		IF uiCommandDoneNum = stAdvHomePara_Set.uiCommandNum THEN//All commands are done
			
			iStep_Homing:=10000;//Done Step
		ELSE
			
			IF uiCommandDoneNum > 0 THEN
				uiCurrentCmdNo:=uiCurrentCmdNo+1;
			END_IF
			
			iStep_Homing:=300;
		END_IF

	300://Decide Step Function and Set Parameter
	
		//Get Homing Para From [SET]
		stAdvHomePara_Local:=stAdvHomePara_Set;
		
		//Set Speed According to Command List content
		IF stAdvHomePara_Local.stHomingCommand[uiCurrentCmdNo].bSlowVelo THEN
			stAdvHomePara_Local.stHomingCommand[uiCurrentCmdNo].stStepFuncParameter.MovePara			:=MovePara_Slow;
			stAdvHomePara_Local.stHomingCommand[uiCurrentCmdNo].stStepFuncParameter.stHomingLimitation	:=MoveLimitation_Slow;
		ELSE
			stAdvHomePara_Local.stHomingCommand[uiCurrentCmdNo].stStepFuncParameter.MovePara			:=MovePara_Fast;
			stAdvHomePara_Local.stHomingCommand[uiCurrentCmdNo].stStepFuncParameter.stHomingLimitation	:=MoveLimitation_Fast;
		END_IF
		
		//Get Homing Function Action Type
		eHome_ActionType:=stAdvHomePara_Local.stHomingCommand[uiCurrentCmdNo].eHome_ActionType;
		
		//Flag On
		IF eHome_ActionType = E_HomingActionType.FinishHoming
		OR eHome_ActionType = E_HomingActionType.HomeDirect 
		THEN
			iStep_FinalizingFunc:=1;
		ELSIF eHome_ActionType = E_HomingActionType.ParameterSetting THEN
			iStep_ParaSetting:=1;
		ELSE
			iStep_StepFunc:=1;
		END_IF
		
		iStep_Homing:=400;
		
	400://Step/Finalizing/Parameter Function
		CASE eHome_ActionType OF
			(* ---------- Step Function ----------*)
			E_HomingActionType.Dog_Abs:
				IF M_DogAbs(stAdvHomePara_Local.stHomingCommand[uiCurrentCmdNo].stStepFuncParameter,lrSetPosition,ErrorId=>uiStepFuncErrorId) THEN
					IF uiStepFuncErrorId = 0 THEN
						uiCommandDoneNum:=uiCommandDoneNum+1;
						iStep_Homing:=200;
					ELSE
						iStep_Homing:=9001;
					END_IF
				END_IF
			E_HomingActionType.Dog_Detection:
				IF M_DogDetection(stAdvHomePara_Local.stHomingCommand[uiCurrentCmdNo].stStepFuncParameter,ErrorId=>uiStepFuncErrorId) THEN
					IF uiStepFuncErrorId = 0 THEN
						uiCommandDoneNum:=uiCommandDoneNum+1;
						iStep_Homing:=200;
					ELSE
						iStep_Homing:=9002;
					END_IF
				END_IF
			E_HomingActionType.Index_Abs:
				IF M_PulseFind(stAdvHomePara_Local.stHomingCommand[uiCurrentCmdNo].stStepFuncParameter,lrSetPosition,ErrorId=>uiStepFuncErrorId) THEN
					IF uiStepFuncErrorId = 0 THEN
						uiCommandDoneNum:=uiCommandDoneNum+1;
						iStep_Homing:=200;
					ELSE
						iStep_Homing:=9003;
					END_IF
				END_IF
			E_HomingActionType.Index_Detection:
				IF M_PulseDetection(stAdvHomePara_Local.stHomingCommand[uiCurrentCmdNo].stStepFuncParameter,ErrorId=>uiStepFuncErrorId) THEN
					IF uiStepFuncErrorId = 0 THEN
						uiCommandDoneNum:=uiCommandDoneNum+1;
						iStep_Homing:=200;
					ELSE
						iStep_Homing:=9004;
					END_IF
				END_IF
			E_HomingActionType.Limit_Abs:
				//Set Ref Switch Signal
				IF stAdvHomePara_Local.bRefNegLimitSignal THEN
					fbStepLimitSwitch.LimitSwitchSignal:=NegLimitSwitchSignal;
				ELSE
					fbStepLimitSwitch.LimitSwitchSignal:=PosLimitSwitchSignal;
				END_IF
				
				IF M_LimitFind(stAdvHomePara_Local.stHomingCommand[uiCurrentCmdNo].stStepFuncParameter,lrSetPosition,ErrorId=>uiStepFuncErrorId) THEN
					IF uiStepFuncErrorId = 0 THEN
						uiCommandDoneNum:=uiCommandDoneNum+1;
						iStep_Homing:=200;
					ELSE
						iStep_Homing:=9005;
					END_IF
				END_IF
			E_HomingActionType.Limit_Detection:
				//Set Ref Switch Signal
				IF stAdvHomePara_Local.bRefNegLimitSignal THEN
					fbStepLimitSwitchDetection.LimitSwitchSignal:=NegLimitSwitchSignal;
				ELSE
					fbStepLimitSwitchDetection.LimitSwitchSignal:=PosLimitSwitchSignal;
				END_IF
				
				IF M_LimitDetection(stAdvHomePara_Local.stHomingCommand[uiCurrentCmdNo].stStepFuncParameter,ErrorId=>uiStepFuncErrorId) THEN
					IF uiStepFuncErrorId = 0 THEN
						uiCommandDoneNum:=uiCommandDoneNum+1;
						iStep_Homing:=200;
					ELSE
						iStep_Homing:=9006;
					END_IF
				END_IF
			(* ---------- Finish Function ----------*)
			E_HomingActionType.FinishHoming:
				IF M_FinishHoming(stAdvHomePara_Local.stHomingCommand[uiCurrentCmdNo].stStepFuncParameter,lrOffset) THEN
					uiCommandDoneNum:=uiCommandDoneNum+1;
					iStep_Homing:=200;
				END_IF
			E_HomingActionType.HomeDirect:
				IF M_HomeDirect(stAdvHomePara_Local.stHomingCommand[uiCurrentCmdNo].stStepFuncParameter,lrSetPosition) THEN
					uiCommandDoneNum:=uiCommandDoneNum+1;
					iStep_Homing:=200;
				END_IF
			(* ---------- Parameter Function ----------*)	
			E_HomingActionType.ParameterSetting:
				IF M_KeepPosBias(stPosBiasPara.bModuloMode,lrSetPosition) THEN
					uiCommandDoneNum:=uiCommandDoneNum+1;
					iStep_Homing:=200;
				END_IF
			E_HomingActionType.MoveAbs:
				IF M_MoveAbs(stAdvHomePara_Local.stHomingCommand[uiCurrentCmdNo].stStepFuncParameter,lrSetPosition) THEN
					IF uiStepFuncErrorId = 0 THEN
						uiCommandDoneNum:=uiCommandDoneNum+1;
						iStep_Homing:=200;
					ELSE
						iStep_Homing:=9007;
					END_IF
				END_IF
			ELSE//Not Defined Action Type
				ErrorId:=400;
				iStep_Homing:=9000;//Error Step
		END_CASE
	
	(*-----Aborting-----*)
	8000://Abort
	
		iStep_FinalizingFunc:=1;
		
		iStep_Homing:=8100;
	8100:
		IF M_AbortHoming() THEN
			iStep_Homing:=10000;
		END_IF
	9000:
		M_SetError(ErrorId);
	(*-----Step Func Error-----*)
	9001..9099:(* Abort *)
		iStep_FinalizingFunc:=1;
		iStep_Homing:=iStep_Homing+100;
	9101..9199:
		IF M_AbortHoming() THEN
			M_SetError(uiStepFuncErrorId);
			iStep_Homing:=iStep_Homing+100;
		END_IF
	(*-----Done-----*)
	10000://Done
		M_SetDone();
		iStep_Homing:=10100;
END_CASE

METHOD PRIVATE M_ClearAllState : BOOL
VAR_INPUT
END_VAR
fbStepAbsoluteSwitchDetection.Execute 	:= FALSE;
fbStepAbsoluteSwitch.Execute 			:= FALSE;				
fbStepLimitSwitchDetection.Execute 		:= FALSE;			
fbStepLimitSwitch.Execute 				:= FALSE;					
fbStepReferencePulse.Execute 			:= FALSE;
fbStepReferencePulseDetection.Execute 	:= FALSE;
fbFinishHoming.Execute					:= FALSE;
fbHomeDirect.Execute					:= FALSE;
fbAbortHoming.Execute 					:= FALSE;

uiCurrentCmdNo:=0;
uiCommandDoneNum:=0;
	
iStep_FinalizingFunc:=0;
iStep_StepFunc:=0;

iStep_Homing:=0;
END_METHOD

METHOD PRIVATE M_ClearSignal : BOOL
VAR_INPUT
END_VAR
Done			:=FALSE;
Busy 			:=FALSE;
Active   		:=FALSE;
CommandAborted	:=FALSE;
Error			:=FALSE;
ErrorId 		:=0;
END_METHOD

METHOD private M_SetBusy : BOOL
VAR_INPUT
END_VAR
M_ClearSignal();

Busy:=TRUE;
END_METHOD

METHOD private M_SetDone : BOOL
VAR_INPUT
END_VAR
M_ClearSignal();

Done:=TRUE;
END_METHOD

METHOD PRIVATE M_SetError : BOOL
VAR_INPUT
	setErrorId:UDINT;
END_VAR
M_ClearSignal();

Error := TRUE;
ErrorId := setErrorId;
END_METHOD

METHOD PRIVATE M_DogAbs : BOOL
VAR_INPUT
	stStepFuncParameter		:ST_StepFuncParameter;
	SetPosition				:LREAL;
END_VAR
VAR_OUTPUT
	ErrorId		:UDINT:=0;
END_VAR
CASE iStep_StepFunc	OF
	1:
		fbStepAbsoluteSwitch.Direction			:= stStepFuncParameter.eHome_Direction;
		fbStepAbsoluteSwitch.SwitchMode		    := stStepFuncParameter.eSwitch_Mode;
		
		fbStepAbsoluteSwitch.Velocity			:= stStepFuncParameter.MovePara.Velocity;
		fbStepAbsoluteSwitch.Acceleration		:= stStepFuncParameter.MovePara.Acc;
		fbStepAbsoluteSwitch.Deceleration		:= stStepFuncParameter.MovePara.Dec;
		fbStepAbsoluteSwitch.Jerk				:= stStepFuncParameter.MovePara.Jerk;
		
		fbStepAbsoluteSwitch.TimeLimit			:= stStepFuncParameter.stHomingLimitation.TimeLimit;
		fbStepAbsoluteSwitch.DistanceLimit		:= stStepFuncParameter.stHomingLimitation.DistanceLimit;
		fbStepAbsoluteSwitch.TorqueLimit		:= stStepFuncParameter.stHomingLimitation.TorqueLimit;
		
		fbStepAbsoluteSwitch.SetPosition		:= SetPosition;
		
		fbStepAbsoluteSwitch.Execute 			:= TRUE;
		
		IF	fbStepAbsoluteSwitch.Busy	THEN
			iStep_StepFunc:= 2;
		END_IF
	
	2:
		IF	fbStepAbsoluteSwitch.Done	THEN
			fbStepAbsoluteSwitch.Execute 		:= FALSE;
			iStep_StepFunc:= 3;	
		ELSIF fbStepAbsoluteSwitch.Error	THEN
			iStep_StepFunc:= 90;
		END_IF
	3:
		iStep_StepFunc:=0;
		M_DogAbs:=TRUE;
	(* Error *)
	90:
		ErrorId:=fbStepAbsoluteSwitch.ErrorID;
		
		fbStepAbsoluteSwitch.Execute:=FALSE;
		M_DogAbs:=TRUE;
END_CASE
END_METHOD

METHOD PRIVATE M_DogDetection : BOOL
VAR_INPUT
	stStepFuncParameter		:ST_StepFuncParameter;
END_VAR
VAR_OUTPUT
	ErrorId		:UDINT:=0;
END_VAR
CASE iStep_StepFunc	OF
	1:
		fbStepAbsoluteSwitchDetection.Direction			:= stStepFuncParameter.eHome_Direction;
		fbStepAbsoluteSwitchDetection.SwitchMode		:= stStepFuncParameter.eSwitch_Mode;
		
		fbStepAbsoluteSwitchDetection.Velocity			:= stStepFuncParameter.MovePara.Velocity;
		fbStepAbsoluteSwitchDetection.Acceleration		:= stStepFuncParameter.MovePara.Acc;
		fbStepAbsoluteSwitchDetection.Deceleration		:= stStepFuncParameter.MovePara.Dec;
		fbStepAbsoluteSwitchDetection.Jerk				:= stStepFuncParameter.MovePara.Jerk;
		
		fbStepAbsoluteSwitchDetection.TimeLimit			:= stStepFuncParameter.stHomingLimitation.TimeLimit;
		fbStepAbsoluteSwitchDetection.DistanceLimit		:= stStepFuncParameter.stHomingLimitation.DistanceLimit;
		fbStepAbsoluteSwitchDetection.TorqueLimit		:= stStepFuncParameter.stHomingLimitation.TorqueLimit;
		
		fbStepAbsoluteSwitchDetection.Execute 			:= TRUE;
		
		IF	fbStepAbsoluteSwitchDetection.Busy	THEN
			iStep_StepFunc:= 2;
		END_IF
	
	2:
		IF	fbStepAbsoluteSwitchDetection.Done	THEN
			fbStepAbsoluteSwitchDetection.Execute 		:= FALSE;
			iStep_StepFunc:= 3;	
		ELSIF fbStepAbsoluteSwitchDetection.Error THEN
			iStep_StepFunc:= 90;
		END_IF
	3:
		iStep_StepFunc:=0;
		M_DogDetection:=TRUE;
	(* Error *)
	90:
		ErrorId:=fbStepAbsoluteSwitchDetection.ErrorID;
		
		fbStepAbsoluteSwitchDetection.Execute:=FALSE;
		M_DogDetection:=TRUE;
END_CASE
END_METHOD

METHOD PRIVATE M_LimitDetection : BOOL
VAR_INPUT
	stStepFuncParameter		:ST_StepFuncParameter;
END_VAR
VAR_OUTPUT
	ErrorId		:UDINT:=0;
END_VAR
CASE iStep_StepFunc	OF
	1:
		fbStepLimitSwitchDetection.Direction			:= stStepFuncParameter.eHome_Direction;
		fbStepLimitSwitchDetection.LimitSwitchMode		:= stStepFuncParameter.eSwitch_Mode;
		
		fbStepLimitSwitchDetection.Velocity			:= stStepFuncParameter.MovePara.Velocity;
		fbStepLimitSwitchDetection.Acceleration		:= stStepFuncParameter.MovePara.Acc;
		fbStepLimitSwitchDetection.Deceleration		:= stStepFuncParameter.MovePara.Dec;
		fbStepLimitSwitchDetection.Jerk				:= stStepFuncParameter.MovePara.Jerk;
		
		fbStepLimitSwitchDetection.TimeLimit		:= stStepFuncParameter.stHomingLimitation.TimeLimit;
		fbStepLimitSwitchDetection.DistanceLimit	:= stStepFuncParameter.stHomingLimitation.DistanceLimit;
		fbStepLimitSwitchDetection.TorqueLimit		:= stStepFuncParameter.stHomingLimitation.TorqueLimit;
		
		fbStepLimitSwitchDetection.Execute := TRUE;
		
		IF	fbStepLimitSwitchDetection.Busy	THEN
			iStep_StepFunc:= 2;
		END_IF
	
	2:
		IF	fbStepLimitSwitchDetection.Done	THEN
			fbStepLimitSwitchDetection.Execute := FALSE;
			iStep_StepFunc:= 3;	
		ELSIF fbStepLimitSwitchDetection.Error THEN
			iStep_StepFunc:= 90;	
		END_IF
	3:
		iStep_StepFunc:=0;
		M_LimitDetection:=TRUE;
	(* Error *)
	90:
		ErrorId:=fbStepLimitSwitchDetection.ErrorID;
		
		fbStepLimitSwitchDetection.Execute:=FALSE;
		M_LimitDetection:=TRUE;
END_CASE
END_METHOD

METHOD PRIVATE M_LimitFind : BOOL
VAR_INPUT
	stStepFuncParameter		:ST_StepFuncParameter;
	SetPosition				:LREAL;
END_VAR
VAR_OUTPUT
	ErrorId		:UDINT:=0;
END_VAR
CASE iStep_StepFunc	OF
	1://拉起找極限
		fbStepLimitSwitch.Direction			:= stStepFuncParameter.eHome_Direction;
		fbStepLimitSwitch.LimitSwitchMode		:= stStepFuncParameter.eSwitch_Mode;
		
		fbStepLimitSwitch.Velocity			:= stStepFuncParameter.MovePara.Velocity;
		fbStepLimitSwitch.Acceleration		:= stStepFuncParameter.MovePara.Acc;
		fbStepLimitSwitch.Deceleration		:= stStepFuncParameter.MovePara.Dec;
		fbStepLimitSwitch.Jerk				:= stStepFuncParameter.MovePara.Jerk;
		
		fbStepLimitSwitch.TimeLimit			:= stStepFuncParameter.stHomingLimitation.TimeLimit;
		fbStepLimitSwitch.DistanceLimit		:= stStepFuncParameter.stHomingLimitation.DistanceLimit;
		fbStepLimitSwitch.TorqueLimit		:= stStepFuncParameter.stHomingLimitation.TorqueLimit;
		
		fbStepLimitSwitch.SetPosition		:= SetPosition;
		
		fbStepLimitSwitch.Execute := TRUE;
		
		IF	fbStepLimitSwitch.Busy	THEN
			iStep_StepFunc:= 2;
		END_IF
	
	2://等待完成
		IF	fbStepLimitSwitch.Done	THEN
			fbStepLimitSwitch.Execute:= FALSE;
			iStep_StepFunc:= 3;	
		ELSIF fbStepLimitSwitch.Error THEN
			iStep_StepFunc:= 90;	
		END_IF
	3://完成處理
		iStep_StepFunc:=0;
		M_LimitFind:=TRUE;
	(* Error *)
	90:
		ErrorId:=fbStepLimitSwitch.ErrorID;
		
		fbStepLimitSwitch.Execute:=FALSE;
		M_LimitFind:=TRUE;
END_CASE
END_METHOD

METHOD M_MoveAbs : BOOL
VAR_INPUT
	stStepFuncParameter		:ST_StepFuncParameter;
	SetPosition				:LREAL;
END_VAR
VAR_OUTPUT
	ErrorId		:UDINT:=0;
END_VAR
CASE iStep_StepFunc OF
    1:
        fbMoveAbs.Acceleration := stStepFuncParameter.MovePara.Acc;
        fbMoveAbs.Deceleration := stStepFuncParameter.MovePara.Dec;
        fbMoveAbs.Jerk := stStepFuncParameter.MovePara.Jerk;
        fbMoveAbs.Velocity := stStepFuncParameter.MovePara.Velocity;
        fbMoveAbs.Position := SetPosition;
		fbMoveAbs.Execute := TRUE;
        IF fbMoveAbs.Busy THEN
            iStep_StepFunc := 2;
        END_IF

    2:
        IF fbMoveAbs.Done THEN
            fbMoveAbs.Execute := FALSE;
            iStep_StepFunc := 3;
        ELSIF fbMoveAbs.Error THEN
            iStep_StepFunc := 90;
        END_IF
    3:
        iStep_StepFunc := 0;
        M_MoveAbs := TRUE;
        (* Error *)
        ErrorId := fbMoveAbs.ErrorID;

        fbMoveAbs.Execute := FALSE;
        M_MoveAbs := TRUE;

END_CASE
END_METHOD

METHOD PRIVATE M_PulseDetection : BOOL
VAR_INPUT
	stStepFuncParameter		:ST_StepFuncParameter;
END_VAR
VAR_OUTPUT
	ErrorId		:UDINT:=0;
END_VAR
CASE iStep_StepFunc	OF
	1:
		fbStepReferencePulseDetection.Direction			:= stStepFuncParameter.eHome_Direction;
		
		fbStepReferencePulseDetection.Velocity			:= stStepFuncParameter.MovePara.Velocity;
		fbStepReferencePulseDetection.Acceleration		:= stStepFuncParameter.MovePara.Acc;
		fbStepReferencePulseDetection.Deceleration		:= stStepFuncParameter.MovePara.Dec;
		fbStepReferencePulseDetection.Jerk				:= stStepFuncParameter.MovePara.Jerk;
		
		fbStepReferencePulseDetection.TimeLimit			:= stStepFuncParameter.stHomingLimitation.TimeLimit;
		fbStepReferencePulseDetection.DistanceLimit		:= stStepFuncParameter.stHomingLimitation.DistanceLimit;
		fbStepReferencePulseDetection.TorqueLimit		:= stStepFuncParameter.stHomingLimitation.TorqueLimit;
		
		fbStepReferencePulseDetection.Execute 			:= TRUE;
		
		IF	fbStepReferencePulseDetection.Busy	THEN
			iStep_StepFunc:= 2;
		END_IF
	
	2:
		IF	fbStepReferencePulseDetection.Done	THEN
			fbStepReferencePulseDetection.Execute 		:= FALSE;
			iStep_StepFunc:= 3;	
		ELSIF fbStepReferencePulseDetection.Error THEN
			iStep_StepFunc:= 90;	
		END_IF
	3:
		iStep_StepFunc:=0;
		M_PulseDetection:=TRUE;
	(* Error *)
	90:
		ErrorId:=fbStepReferencePulseDetection.ErrorID;
		
		fbStepReferencePulseDetection.Execute:=FALSE;
		M_PulseDetection:=TRUE;
END_CASE
END_METHOD

METHOD PRIVATE M_PulseFind : BOOL
VAR_INPUT
	stStepFuncParameter		:ST_StepFuncParameter;
	SetPosition				:LREAL;
END_VAR
VAR_OUTPUT
	ErrorId		:UDINT:=0;
END_VAR
CASE iStep_StepFunc OF 
	1://拉起找Zero Pulse
	
		fbStepReferencePulse.Direction			:= stStepFuncParameter.eHome_Direction;
		
		fbStepReferencePulse.Velocity			:= stStepFuncParameter.MovePara.Velocity;
		fbStepReferencePulse.Acceleration		:= stStepFuncParameter.MovePara.Acc;
		fbStepReferencePulse.Deceleration		:= stStepFuncParameter.MovePara.Dec;
		fbStepReferencePulse.Jerk				:= stStepFuncParameter.MovePara.Jerk;
		
		fbStepReferencePulse.TimeLimit			:= stStepFuncParameter.stHomingLimitation.TimeLimit;
		fbStepReferencePulse.DistanceLimit		:= stStepFuncParameter.stHomingLimitation.DistanceLimit;
		fbStepReferencePulse.TorqueLimit		:= stStepFuncParameter.stHomingLimitation.TorqueLimit;
		
		fbStepReferencePulse.SetPosition		:= SetPosition;
		
		fbStepReferencePulse.Execute 			:= TRUE;
		
		IF	fbStepReferencePulse.Busy THEN
			iStep_StepFunc:= 2;
		END_IF
	
	2:
		IF	fbStepReferencePulse.Done	THEN
			fbStepReferencePulse.Execute:= FALSE;
			iStep_StepFunc:= 3;
		ELSIF fbStepReferencePulse.Error THEN
			iStep_StepFunc:= 90;
		END_IF
	3:
		iStep_StepFunc:=0;
		M_PulseFind:=TRUE;
	(* Error *)
	90:
		ErrorId:=fbStepReferencePulse.ErrorID;
		
		fbStepReferencePulse.Execute:=FALSE;
		M_PulseFind:=TRUE;
END_CASE
END_METHOD

METHOD PRIVATE M_AbortHoming : BOOL
VAR_INPUT
END_VAR
CASE iStep_FinalizingFunc OF
	1:
		fbAbortHoming.Execute 					:= TRUE;
		
		IF	fbAbortHoming.Busy	THEN
			iStep_FinalizingFunc:= 2;
		END_IF
	2:
		IF	fbAbortHoming.Done	THEN
			fbAbortHoming.Execute 		:= FALSE;
			iStep_FinalizingFunc:= 3;	
		END_IF
	3:
		iStep_FinalizingFunc:=0;
		M_AbortHoming:=TRUE;
END_CASE
END_METHOD

METHOD PRIVATE M_FinishHoming : BOOL
VAR_INPUT
	stStepFuncParameter		:ST_StepFuncParameter;
	Distance				:LREAL;
END_VAR
CASE iStep_FinalizingFunc OF
	1:
		fbFinishHoming.Velocity			:= stStepFuncParameter.MovePara.Velocity;
		fbFinishHoming.Acceleration		:= stStepFuncParameter.MovePara.Acc;
		fbFinishHoming.Deceleration		:= stStepFuncParameter.MovePara.Dec;
		fbFinishHoming.Jerk				:= stStepFuncParameter.MovePara.Jerk;
		
		fbFinishHoming.Distance			:=Distance;
		
		fbFinishHoming.Execute 			:= TRUE;
		
		IF	fbFinishHoming.Busy	THEN
			iStep_FinalizingFunc:= 2;
		END_IF
	2:
		IF	fbFinishHoming.Done	THEN
			fbFinishHoming.Execute 		:= FALSE;
			iStep_FinalizingFunc:= 3;	
		END_IF
	3:
		iStep_FinalizingFunc:=0;
		M_FinishHoming:=TRUE;
END_CASE
END_METHOD

METHOD PRIVATE M_HomeDirect : BOOL
VAR_INPUT
	stStepFuncParameter		:ST_StepFuncParameter;
	SetPosition				:LREAL;
END_VAR
CASE iStep_FinalizingFunc OF
	1:
		fbHomeDirect.SetPosition:=SetPosition;
		
		fbHomeDirect.Execute:=TRUE;
		
		IF	fbHomeDirect.Busy	THEN
			iStep_FinalizingFunc:= 2;
		END_IF
	2:
		IF	fbHomeDirect.Done	THEN
			fbHomeDirect.Execute 		:= FALSE;
			iStep_FinalizingFunc:= 3;	
		END_IF
	3:
		iStep_FinalizingFunc:=0;
		M_HomeDirect:=TRUE;
END_CASE
END_METHOD

METHOD M_KeepPosBias : BOOL
VAR_INPUT
	bModuloMode		:BOOL:=FALSE;//True=Modulo Bias
	SetPosition		:LREAL;
END_VAR
VAR
	lrNcCurrentBias	:LREAL;
	lrNcCurrentPos	:LREAL;
	lrNcTargetPos	:LREAL;
	lrNcTargetBias	:LREAL;
	lrNcOriginPos	:LREAL;
END_VAR
CASE iStep_ParaSetting OF
	1://Read Current Bias Value
	
		fbReadParameter.Enable				:= TRUE;
		fbReadParameter.ReadMode			:= E_ReadMode.READMODE_ONCE;
		fbReadParameter.ParameterNumber		:= MC_AxisParameter.AxisEncoderOffset;//Position Bias
		
		IF fbReadParameter.Valid THEN
			fbReadParameter.Enable:=FALSE;
			iStep_ParaSetting:= 2;
		ELSIF fbReadParameter.Error THEN
			;
		END_IF
	2://Set Position Bias
	
		//Current Value
		IF bModuloMode THEN
			lrNcCurrentPos 	:= THIS^.AxisRef.NcToPlc.ModuloActPos;
		ELSE
			lrNcCurrentPos 	:= THIS^.AxisRef.NcToPlc.ActPos;
		END_IF
		
		lrNcCurrentBias	:= fbReadParameter.Value;
		
		//當前座標 - 已經套用的Bias = 原始座標
		////lrNcOriginPos	:= lrNcCurrentPos - THIS^.refNcPositionBias;
		lrNcOriginPos	:= lrNcCurrentPos - THIS^.refAxisPara.stPositionBias_Ctrl.lrPosBiasValue;
		
		//New Value
		lrNcTargetPos			:= SetPosition;	
		lrNcTargetBias			:= lrNcTargetPos - lrNcOriginPos;	//要設定的Target座標 - 原始座標 = 完整的Bias
		
		//Output to Ref Var(Persistent)
		THIS^.lrPosBiasValue	:= lrNcTargetBias;		
		
		iStep_ParaSetting:= 0;
		M_KeepPosBias			:=TRUE;
	(*
	3://Write Persistent
	
		//Write Persistent
		fbWritePersistent.PORT	:= 851;
		fbWritePersistent.START	:= TRUE;
		
		IF NOT fbWritePersistent.BUSY AND NOT fbWritePersistent.ERR THEN
			fbWritePersistent.START	:= FALSE;
			iStep_ParaSetting		:=0;
			M_KeepPosBias			:=TRUE;
		ELSIF fbWritePersistent.ERR THEN
			;
		END_IF
	*)
END_CASE
END_METHOD

ACTION A_ActionTrigger:
rTrig_Start(CLK:=bStartHoming);
fTrig_Start(CLK:=bStartHoming);
rTrig_Abort(CLK:=bAbortHoming);
fTrig_Abort(CLK:=bAbortHoming);

//Start Homing
IF rTrig_Start.Q THEN
	
	M_ClearAllState();

	M_SetBusy();
	
	iStep_Homing:=100;
END_IF

IF fTrig_Start.Q THEN
	M_ClearAllState();
	M_ClearSignal();
END_IF

//Abort Homing
IF rTrig_Abort.Q THEN
	
	M_ClearAllState();
	
	M_SetBusy();
	
	iStep_Homing:=8000;
END_IF

IF fTrig_Abort.Q THEN
	M_ClearAllState();
	M_ClearSignal();
END_IF
END_ACTION

ACTION A_CyclicUpdate:
(* ----------Signal Refresh----------*)
//Di Signal
DogSignal.Level				:=bDogSignal;
PosLimitSwitchSignal.Level	:=bPosLimitSignal;
NegLimitSwitchSignal.Level	:=bNegLimitSignal;
//Index
IF bSimuMode THEN
	ZeroSwitchSignal.Level			:=ZeroSwitchSignal.Level;
	ZeroSwitchSignal.SignalSource	:=E_SignalSource.SignalSource_Default;
	ZeroSwitchSignal.TouchProbe		:=E_TouchProbe.PlcEvent;
ELSE
	ZeroSwitchSignal.Level			:=ZeroSwitchSignal.Level;
	ZeroSwitchSignal.SignalSource	:=E_SignalSource.SignalSource_ZeroPulse;
	ZeroSwitchSignal.TouchProbe		:=E_TouchProbe.TouchProbe1;
END_IF


(* ----------Parameter Refresh----------*)
IF bThirdPartyDrive OR bSimuMode THEN
	Options2.DisableDriveAccess	:= TRUE;
	Options4.DisableDriveAccess	:= TRUE;
ELSE
	Options2.DisableDriveAccess	:= FALSE;
	Options4.DisableDriveAccess	:= FALSE;
END_IF

fbStepReferencePulse.ReferenceSignal				:=ZeroSwitchSignal;
fbStepReferencePulseDetection.ReferenceSignal		:=ZeroSwitchSignal;

fbStepAbsoluteSwitch.ReferenceSignal				:=DogSignal;
fbStepAbsoluteSwitchDetection.ReferenceSignal		:=DogSignal;

fbStepAbsoluteSwitch.PositiveLimitSwitch			:=bPosLimitSignal;
fbStepAbsoluteSwitchDetection.PositiveLimitSwitch	:=bPosLimitSignal;

fbStepAbsoluteSwitch.NegativeLimitSwitch			:=bNegLimitSignal;
fbStepAbsoluteSwitchDetection.NegativeLimitSwitch	:=bNegLimitSignal;

(* ----------FB Refresh----------*)
//Step Function
fbStepAbsoluteSwitchDetection(Axis := AxisRef ,Parameter := Parameter, Options := Options4);

fbStepAbsoluteSwitch(Axis := AxisRef, Parameter := Parameter, Options := Options4);

fbStepLimitSwitchDetection(Axis := AxisRef, Parameter := Parameter, Options := Options4);
		
fbStepLimitSwitch(Axis := AxisRef, Parameter := Parameter, Options := Options4);

fbStepReferencePulse(Axis := AxisRef, Parameter := Parameter, Options := Options4);

fbStepReferencePulseDetection(Axis := AxisRef, Parameter := Parameter, Options := Options4);

//Finalizing Function
fbFinishHoming(Axis := AxisRef, Parameter := Parameter, Options := Options2);
		
fbHomeDirect(Axis := AxisRef, Parameter := Parameter, Options := Options2);

fbAbortHoming(Axis := AxisRef, Parameter := Parameter, Options := Options2);

//NC Parameter
fbReadParameter(Axis:= AxisRef);
END_ACTION

METHOD M_CheckSignalConnected : BOOL
VAR_INPUT
	edHomingMode:E_HomingMode;
END_VAR
VAR
	wSiganlBit_Connected:WORD:=0;
	wSiganlBit_Check	:WORD:=0;
	
	wDog				:WORD:=2#001;
	wPosLimit			:WORD:=2#010;
	wNegLimit			:WORD:=2#100;
		
END_VAR
IF bDogConnected THEN
	wSiganlBit_Connected:=(wSiganlBit_Connected OR wDog);//2^0
END_IF
IF bPosLimitConnected THEN
	wSiganlBit_Connected:=(wSiganlBit_Connected OR wPosLimit);//2^1
END_IF
IF bNegLimitConnected THEN
	wSiganlBit_Connected:=(wSiganlBit_Connected OR wNegLimit);//2^2
END_IF

CASE edHomingMode OF
	E_HomingMode._01_Neg_LimitOutterRightIndex:				wSiganlBit_Check:=(wNegLimit);
	E_HomingMode._02_Pos_LimitOutterLeftIndex:				wSiganlBit_Check:=(wPosLimit);
	E_HomingMode._03_Pos_HomeOutterLeftIndex:				wSiganlBit_Check:=(wDog);
	E_HomingMode._04_Pos_HomeInnerLeftIndex:				wSiganlBit_Check:=(wDog);
	E_HomingMode._05_Neg_HomeOutterRightIndex:				wSiganlBit_Check:=(wDog);
	E_HomingMode._06_Neg_HomeInnerRightIndex:				wSiganlBit_Check:=(wDog);
	E_HomingMode._07_Pos_HomeOutterLeftIndex_withLimit:		wSiganlBit_Check:=(wDog OR wPosLimit OR wNegLimit);
	E_HomingMode._08_Pos_HomeInnerLeftIndex_withLimit:		wSiganlBit_Check:=(wDog OR wPosLimit OR wNegLimit);
	E_HomingMode._09_Pos_HomeInnerRightIndex_withLimit:		wSiganlBit_Check:=(wDog OR wPosLimit OR wNegLimit);
	E_HomingMode._10_Pos_HomeOutterRightIndex_withLimit:	wSiganlBit_Check:=(wDog OR wPosLimit OR wNegLimit);
	E_HomingMode._11_Neg_HomeOutterRightIndex_withLimit:	wSiganlBit_Check:=(wDog OR wPosLimit OR wNegLimit);
	E_HomingMode._12_Neg_HomeInnerRightIndex_withLimit:		wSiganlBit_Check:=(wDog OR wPosLimit OR wNegLimit);
	E_HomingMode._13_Neg_HomeInnerLeftIndex_withLimit:		wSiganlBit_Check:=(wDog OR wPosLimit OR wNegLimit);
	E_HomingMode._14_Neg_HomeOutterLeftIndex_withLimit:		wSiganlBit_Check:=(wDog OR wPosLimit OR wNegLimit);
	E_HomingMode._17_Neg_LimitOutterRight:					wSiganlBit_Check:=(wNegLimit);
	E_HomingMode._18_Pos_LimitOutterLeft:					wSiganlBit_Check:=(wPosLimit);
	E_HomingMode._19_Pos_HomeOutterLeft:					wSiganlBit_Check:=(wDog);
	E_HomingMode._20_Pos_HomeInnerLeft:						wSiganlBit_Check:=(wDog);
	E_HomingMode._21_Neg_HomeOutterRight:					wSiganlBit_Check:=(wDog);
	E_HomingMode._22_Neg_HomeInnerRight:					wSiganlBit_Check:=(wDog);
	E_HomingMode._23_Pos_HomeOutterLeft_withLimit:			wSiganlBit_Check:=(wDog OR wPosLimit OR wNegLimit);
	E_HomingMode._24_Pos_HomeInnerLeft_withLimit:			wSiganlBit_Check:=(wDog OR wPosLimit OR wNegLimit);
	E_HomingMode._25_Pos_HomeInnerRight_withLimit:			wSiganlBit_Check:=(wDog OR wPosLimit OR wNegLimit);
	E_HomingMode._26_Pos_HomeOutterRight_withLimit:			wSiganlBit_Check:=(wDog OR wPosLimit OR wNegLimit);
	E_HomingMode._27_Neg_HomeOutterRight_withLimit:			wSiganlBit_Check:=(wDog OR wPosLimit OR wNegLimit);
	E_HomingMode._28_Neg_HomeInnerRight_withLimit:			wSiganlBit_Check:=(wDog OR wPosLimit OR wNegLimit);
	E_HomingMode._29_Neg_HomeInnerLeft_withLimit:			wSiganlBit_Check:=(wDog OR wPosLimit OR wNegLimit);
	E_HomingMode._30_Neg_HomeOutterLeft_withLimit:			wSiganlBit_Check:=(wDog OR wPosLimit OR wNegLimit);
	E_HomingMode._33_Neg_Index:								wSiganlBit_Check:=0;
	E_HomingMode._34_Pos_Index:								wSiganlBit_Check:=0;
	E_HomingMode._35_CurrentPosition:						wSiganlBit_Check:=0;
END_CASE

IF (wSiganlBit_Connected AND wSiganlBit_Check) = wSiganlBit_Check THEN
	M_CheckSignalConnected:=TRUE;
ELSE
	M_CheckSignalConnected:=FALSE;
END_IF
END_METHOD

METHOD M_SelectPreDefinedMode : BOOL
VAR_INPUT
	udHomingMode		:E_HomingMode;
	bSetPostionBias		:BOOL;
END_VAR
//Clear Old Parameter
stAdvHomePara_Set := stAdvHomePara_Clear;

CASE udHomingMode OF
    E_HomingMode._01_Neg_LimitOutterRightIndex:

        //Ref Limit Siganl
        stAdvHomePara_Set.bRefNegLimitSignal := TRUE;

        //Find Limit -
        stAdvHomePara_Set.stHomingCommand[0].eHome_ActionType := E_HomingActionType.Limit_Detection;
        stAdvHomePara_Set.stHomingCommand[0].bSlowVelo := FALSE;
        stAdvHomePara_Set.stHomingCommand[0].stStepFuncParameter.eHome_Direction := MC_Home_Direction.mcNegativeDirection;
        stAdvHomePara_Set.stHomingCommand[0].stStepFuncParameter.eSwitch_Mode := MC_Switch_Mode.mcOn;

        //Escape from Limit
        stAdvHomePara_Set.stHomingCommand[1].eHome_ActionType := E_HomingActionType.Limit_Detection;
        stAdvHomePara_Set.stHomingCommand[1].bSlowVelo := TRUE;
        stAdvHomePara_Set.stHomingCommand[1].stStepFuncParameter.eHome_Direction := MC_Home_Direction.mcNegativeDirection;
        stAdvHomePara_Set.stHomingCommand[1].stStepFuncParameter.eSwitch_Mode := MC_Switch_Mode.mcFallingEdge;

        //Pos Find Pulse
        stAdvHomePara_Set.stHomingCommand[2].eHome_ActionType := E_HomingActionType.Index_Detection;
        stAdvHomePara_Set.stHomingCommand[2].bSlowVelo := TRUE;
        stAdvHomePara_Set.stHomingCommand[2].stStepFuncParameter.eHome_Direction := MC_Home_Direction.mcPositiveDirection;

        //Shift Distance
        stAdvHomePara_Set.stHomingCommand[3].eHome_ActionType := E_HomingActionType.FinishHoming;
        stAdvHomePara_Set.stHomingCommand[3].bSlowVelo := TRUE;

        IF NOT bSetPostionBias THEN

            //Set Position
            stAdvHomePara_Set.stHomingCommand[4].eHome_ActionType := E_HomingActionType.HomeDirect;

            stAdvHomePara_Set.uiCommandNum := 5;
        ELSE
            //Set Bias
            stAdvHomePara_Set.stHomingCommand[4].eHome_ActionType := E_HomingActionType.ParameterSetting;

            //Set Position
            stAdvHomePara_Set.stHomingCommand[5].eHome_ActionType := E_HomingActionType.HomeDirect;

            stAdvHomePara_Set.uiCommandNum := 6;
        END_IF

    E_HomingMode._02_Pos_LimitOutterLeftIndex:

        //Ref Limit Siganl
        stAdvHomePara_Set.bRefNegLimitSignal := FALSE;

        //Find Limit +
        stAdvHomePara_Set.stHomingCommand[0].eHome_ActionType := E_HomingActionType.Limit_Detection;
        stAdvHomePara_Set.stHomingCommand[0].bSlowVelo := FALSE;
        stAdvHomePara_Set.stHomingCommand[0].stStepFuncParameter.eHome_Direction := MC_Home_Direction.mcPositiveDirection;
        stAdvHomePara_Set.stHomingCommand[0].stStepFuncParameter.eSwitch_Mode := MC_Switch_Mode.mcOn;

        //Escape from Limit
        stAdvHomePara_Set.stHomingCommand[1].eHome_ActionType := E_HomingActionType.Limit_Detection;
        stAdvHomePara_Set.stHomingCommand[1].bSlowVelo := TRUE;
        stAdvHomePara_Set.stHomingCommand[1].stStepFuncParameter.eHome_Direction := MC_Home_Direction.mcPositiveDirection;
        stAdvHomePara_Set.stHomingCommand[1].stStepFuncParameter.eSwitch_Mode := MC_Switch_Mode.mcFallingEdge;

        //Neg Find Pulse
        stAdvHomePara_Set.stHomingCommand[2].eHome_ActionType := E_HomingActionType.Index_Detection;
        stAdvHomePara_Set.stHomingCommand[2].bSlowVelo := TRUE;
        stAdvHomePara_Set.stHomingCommand[2].stStepFuncParameter.eHome_Direction := MC_Home_Direction.mcNegativeDirection;

        //Shift Distance
        stAdvHomePara_Set.stHomingCommand[3].eHome_ActionType := E_HomingActionType.FinishHoming;
        stAdvHomePara_Set.stHomingCommand[3].bSlowVelo := TRUE;

        IF NOT bSetPostionBias THEN

            //Set Position
            stAdvHomePara_Set.stHomingCommand[4].eHome_ActionType := E_HomingActionType.HomeDirect;

            stAdvHomePara_Set.uiCommandNum := 5;

        ELSE
            //Set Bias
            stAdvHomePara_Set.stHomingCommand[4].eHome_ActionType := E_HomingActionType.ParameterSetting;

            //Set Position
            stAdvHomePara_Set.stHomingCommand[5].eHome_ActionType := E_HomingActionType.HomeDirect;

            stAdvHomePara_Set.uiCommandNum := 6;
        END_IF

    E_HomingMode._03_Pos_HomeOutterLeftIndex: //Done

        //Find Home +
        stAdvHomePara_Set.stHomingCommand[0].eHome_ActionType := E_HomingActionType.Dog_Detection;
        stAdvHomePara_Set.stHomingCommand[0].bSlowVelo := FALSE;
        stAdvHomePara_Set.stHomingCommand[0].stStepFuncParameter.eHome_Direction := MC_Home_Direction.mcPositiveDirection;
        stAdvHomePara_Set.stHomingCommand[0].stStepFuncParameter.eSwitch_Mode := MC_Switch_Mode.mcOn;

        //Neg Escpape From Home
        stAdvHomePara_Set.stHomingCommand[1].eHome_ActionType := E_HomingActionType.Dog_Detection;
        stAdvHomePara_Set.stHomingCommand[1].bSlowVelo := TRUE;
        stAdvHomePara_Set.stHomingCommand[1].stStepFuncParameter.eHome_Direction := MC_Home_Direction.mcNegativeDirection;
        stAdvHomePara_Set.stHomingCommand[1].stStepFuncParameter.eSwitch_Mode := MC_Switch_Mode.mcFallingEdge;

        //Neg Find Pulse
        stAdvHomePara_Set.stHomingCommand[2].eHome_ActionType := E_HomingActionType.Index_Detection;
        stAdvHomePara_Set.stHomingCommand[2].bSlowVelo := TRUE;
        stAdvHomePara_Set.stHomingCommand[2].stStepFuncParameter.eHome_Direction := MC_Home_Direction.mcNegativeDirection;

        //Shift Distance
        stAdvHomePara_Set.stHomingCommand[3].eHome_ActionType := E_HomingActionType.FinishHoming;
        stAdvHomePara_Set.stHomingCommand[3].bSlowVelo := TRUE;

        IF NOT bSetPostionBias THEN
            //Set Position
            stAdvHomePara_Set.stHomingCommand[4].eHome_ActionType := E_HomingActionType.HomeDirect;

            stAdvHomePara_Set.uiCommandNum := 5;
        ELSE
            //Set Bias
            stAdvHomePara_Set.stHomingCommand[4].eHome_ActionType := E_HomingActionType.ParameterSetting;

            //Set Position
            stAdvHomePara_Set.stHomingCommand[5].eHome_ActionType := E_HomingActionType.HomeDirect;

            stAdvHomePara_Set.uiCommandNum := 6;
        END_IF

    E_HomingMode._04_Pos_HomeInnerLeftIndex:

        //Find Home +
        stAdvHomePara_Set.stHomingCommand[0].eHome_ActionType := E_HomingActionType.Dog_Detection;
        stAdvHomePara_Set.stHomingCommand[0].bSlowVelo := FALSE;
        stAdvHomePara_Set.stHomingCommand[0].stStepFuncParameter.eHome_Direction := MC_Home_Direction.mcPositiveDirection;
        stAdvHomePara_Set.stHomingCommand[0].stStepFuncParameter.eSwitch_Mode := MC_Switch_Mode.mcOn;

        //Escape from Home and Re-Enter
        stAdvHomePara_Set.stHomingCommand[1].eHome_ActionType := E_HomingActionType.Dog_Detection;
        stAdvHomePara_Set.stHomingCommand[1].bSlowVelo := TRUE;
        stAdvHomePara_Set.stHomingCommand[1].stStepFuncParameter.eHome_Direction := MC_Home_Direction.mcSwitchPositive;
        stAdvHomePara_Set.stHomingCommand[1].stStepFuncParameter.eSwitch_Mode := MC_Switch_Mode.mcRisingEdge;

        //Pos Find Pulse
        stAdvHomePara_Set.stHomingCommand[2].eHome_ActionType := E_HomingActionType.Index_Detection;
        stAdvHomePara_Set.stHomingCommand[2].bSlowVelo := TRUE;
        stAdvHomePara_Set.stHomingCommand[2].stStepFuncParameter.eHome_Direction := MC_Home_Direction.mcPositiveDirection;

        //Shift Distance
        stAdvHomePara_Set.stHomingCommand[3].eHome_ActionType := E_HomingActionType.FinishHoming;
        stAdvHomePara_Set.stHomingCommand[3].bSlowVelo := TRUE;

        IF NOT bSetPostionBias THEN
            //Set Position
            stAdvHomePara_Set.stHomingCommand[4].eHome_ActionType := E_HomingActionType.HomeDirect;

            stAdvHomePara_Set.uiCommandNum := 5;
        ELSE
            //Set Bias
            stAdvHomePara_Set.stHomingCommand[4].eHome_ActionType := E_HomingActionType.ParameterSetting;

            //Set Position
            stAdvHomePara_Set.stHomingCommand[5].eHome_ActionType := E_HomingActionType.HomeDirect;

            stAdvHomePara_Set.uiCommandNum := 6;
        END_IF

    E_HomingMode._05_Neg_HomeOutterRightIndex: //Done

        //Find Home -
        stAdvHomePara_Set.stHomingCommand[0].eHome_ActionType := E_HomingActionType.Dog_Detection;
        stAdvHomePara_Set.stHomingCommand[0].bSlowVelo := FALSE;
        stAdvHomePara_Set.stHomingCommand[0].stStepFuncParameter.eHome_Direction := MC_Home_Direction.mcNegativeDirection;
        stAdvHomePara_Set.stHomingCommand[0].stStepFuncParameter.eSwitch_Mode := MC_Switch_Mode.mcOn;

        //Escape from Limit 
        stAdvHomePara_Set.stHomingCommand[1].eHome_ActionType := E_HomingActionType.Dog_Detection;
        stAdvHomePara_Set.stHomingCommand[1].bSlowVelo := TRUE;
        stAdvHomePara_Set.stHomingCommand[1].stStepFuncParameter.eHome_Direction := MC_Home_Direction.mcPositiveDirection;
        stAdvHomePara_Set.stHomingCommand[1].stStepFuncParameter.eSwitch_Mode := MC_Switch_Mode.mcFallingEdge;

        //Pos Find Pulse +
        stAdvHomePara_Set.stHomingCommand[2].eHome_ActionType := E_HomingActionType.Index_Detection;
        stAdvHomePara_Set.stHomingCommand[2].bSlowVelo := TRUE;
        stAdvHomePara_Set.stHomingCommand[2].stStepFuncParameter.eHome_Direction := MC_Home_Direction.mcPositiveDirection;

        //Shift Distance
        stAdvHomePara_Set.stHomingCommand[3].eHome_ActionType := E_HomingActionType.FinishHoming;
        stAdvHomePara_Set.stHomingCommand[3].bSlowVelo := TRUE;

        IF NOT bSetPostionBias THEN
            //Set Position
            stAdvHomePara_Set.stHomingCommand[4].eHome_ActionType := E_HomingActionType.HomeDirect;

            stAdvHomePara_Set.uiCommandNum := 5;
        ELSE
            //Set Bias
            stAdvHomePara_Set.stHomingCommand[4].eHome_ActionType := E_HomingActionType.ParameterSetting;

            //Set Position
            stAdvHomePara_Set.stHomingCommand[5].eHome_ActionType := E_HomingActionType.HomeDirect;

            stAdvHomePara_Set.uiCommandNum := 6;
        END_IF

    E_HomingMode._06_Neg_HomeInnerRightIndex:

        //Find Home -
        stAdvHomePara_Set.stHomingCommand[0].eHome_ActionType := E_HomingActionType.Dog_Detection;
        stAdvHomePara_Set.stHomingCommand[0].bSlowVelo := FALSE;
        stAdvHomePara_Set.stHomingCommand[0].stStepFuncParameter.eHome_Direction := MC_Home_Direction.mcSwitchNegative;
        stAdvHomePara_Set.stHomingCommand[0].stStepFuncParameter.eSwitch_Mode := MC_Switch_Mode.mcOn;

        //Escape from Home and Re-Enter
        stAdvHomePara_Set.stHomingCommand[1].eHome_ActionType := E_HomingActionType.Dog_Detection;
        stAdvHomePara_Set.stHomingCommand[1].bSlowVelo := TRUE;
        stAdvHomePara_Set.stHomingCommand[1].stStepFuncParameter.eHome_Direction := MC_Home_Direction.mcSwitchNegative;
        stAdvHomePara_Set.stHomingCommand[1].stStepFuncParameter.eSwitch_Mode := MC_Switch_Mode.mcRisingEdge;

        //Neg Find Pulse
        stAdvHomePara_Set.stHomingCommand[2].eHome_ActionType := E_HomingActionType.Index_Detection;
        stAdvHomePara_Set.stHomingCommand[2].bSlowVelo := TRUE;
        stAdvHomePara_Set.stHomingCommand[2].stStepFuncParameter.eHome_Direction := MC_Home_Direction.mcNegativeDirection;

        //Shift Distance
        stAdvHomePara_Set.stHomingCommand[3].eHome_ActionType := E_HomingActionType.FinishHoming;
        stAdvHomePara_Set.stHomingCommand[3].bSlowVelo := TRUE;

        IF NOT bSetPostionBias THEN

            //Set Position
            stAdvHomePara_Set.stHomingCommand[4].eHome_ActionType := E_HomingActionType.HomeDirect;

            stAdvHomePara_Set.uiCommandNum := 5;

        ELSE
            //Set Bias
            stAdvHomePara_Set.stHomingCommand[4].eHome_ActionType := E_HomingActionType.ParameterSetting;

            //Set Position
            stAdvHomePara_Set.stHomingCommand[5].eHome_ActionType := E_HomingActionType.HomeDirect;

            stAdvHomePara_Set.uiCommandNum := 6;
        END_IF

    E_HomingMode._07_Pos_HomeOutterLeftIndex_withLimit: //Done

        //Pos Find Home
        stAdvHomePara_Set.stHomingCommand[0].eHome_ActionType := E_HomingActionType.Dog_Detection;
        stAdvHomePara_Set.stHomingCommand[0].bSlowVelo := FALSE;
        stAdvHomePara_Set.stHomingCommand[0].stStepFuncParameter.eHome_Direction := MC_Home_Direction.mcPositiveDirection;
        stAdvHomePara_Set.stHomingCommand[0].stStepFuncParameter.eSwitch_Mode := MC_Switch_Mode.mcOn;

        //Neg Escape from Home
        stAdvHomePara_Set.stHomingCommand[1].eHome_ActionType := E_HomingActionType.Dog_Detection;
        stAdvHomePara_Set.stHomingCommand[1].bSlowVelo := TRUE;
        stAdvHomePara_Set.stHomingCommand[1].stStepFuncParameter.eHome_Direction := MC_Home_Direction.mcNegativeDirection;
        stAdvHomePara_Set.stHomingCommand[1].stStepFuncParameter.eSwitch_Mode := MC_Switch_Mode.mcFallingEdge;

        //Neg Find Pulse
        stAdvHomePara_Set.stHomingCommand[2].eHome_ActionType := E_HomingActionType.Index_Detection;
        stAdvHomePara_Set.stHomingCommand[2].bSlowVelo := TRUE;
        stAdvHomePara_Set.stHomingCommand[2].stStepFuncParameter.eHome_Direction := MC_Home_Direction.mcNegativeDirection;

        //Shift Distance
        stAdvHomePara_Set.stHomingCommand[3].eHome_ActionType := E_HomingActionType.FinishHoming;
        stAdvHomePara_Set.stHomingCommand[3].bSlowVelo := TRUE;

        IF NOT bSetPostionBias THEN

            //Set Position
            stAdvHomePara_Set.stHomingCommand[4].eHome_ActionType := E_HomingActionType.HomeDirect;

            stAdvHomePara_Set.uiCommandNum := 5;

        ELSE
            //Set Bias
            stAdvHomePara_Set.stHomingCommand[4].eHome_ActionType := E_HomingActionType.ParameterSetting;

            //Set Position
            stAdvHomePara_Set.stHomingCommand[5].eHome_ActionType := E_HomingActionType.HomeDirect;

            stAdvHomePara_Set.uiCommandNum := 6;
        END_IF

    E_HomingMode._08_Pos_HomeInnerLeftIndex_withLimit:

        //Find Home +
        stAdvHomePara_Set.stHomingCommand[0].eHome_ActionType := E_HomingActionType.Dog_Detection;
        stAdvHomePara_Set.stHomingCommand[0].bSlowVelo := FALSE;
        stAdvHomePara_Set.stHomingCommand[0].stStepFuncParameter.eHome_Direction := MC_Home_Direction.mcPositiveDirection;
        stAdvHomePara_Set.stHomingCommand[0].stStepFuncParameter.eSwitch_Mode := MC_Switch_Mode.mcOn;

        //Escape from Home and Re-Enter
        stAdvHomePara_Set.stHomingCommand[1].eHome_ActionType := E_HomingActionType.Dog_Detection;
        stAdvHomePara_Set.stHomingCommand[1].bSlowVelo := TRUE;
        stAdvHomePara_Set.stHomingCommand[1].stStepFuncParameter.eHome_Direction := MC_Home_Direction.mcSwitchPositive;
        stAdvHomePara_Set.stHomingCommand[1].stStepFuncParameter.eSwitch_Mode := MC_Switch_Mode.mcRisingEdge;

        //Pos Find Pulse
        stAdvHomePara_Set.stHomingCommand[2].eHome_ActionType := E_HomingActionType.Index_Detection;
        stAdvHomePara_Set.stHomingCommand[2].bSlowVelo := TRUE;
        stAdvHomePara_Set.stHomingCommand[2].stStepFuncParameter.eHome_Direction := MC_Home_Direction.mcPositiveDirection;

        //Shift Distance
        stAdvHomePara_Set.stHomingCommand[3].eHome_ActionType := E_HomingActionType.FinishHoming;
        stAdvHomePara_Set.stHomingCommand[3].bSlowVelo := TRUE;

        IF NOT bSetPostionBias THEN

            //Set Position
            stAdvHomePara_Set.stHomingCommand[4].eHome_ActionType := E_HomingActionType.HomeDirect;

            stAdvHomePara_Set.uiCommandNum := 5;

        ELSE
            //Set Bias
            stAdvHomePara_Set.stHomingCommand[4].eHome_ActionType := E_HomingActionType.ParameterSetting;

            //Set Position
            stAdvHomePara_Set.stHomingCommand[5].eHome_ActionType := E_HomingActionType.HomeDirect;

            stAdvHomePara_Set.uiCommandNum := 6;
        END_IF

    E_HomingMode._09_Pos_HomeInnerRightIndex_withLimit:

        //Find Home +
        stAdvHomePara_Set.stHomingCommand[0].eHome_ActionType := E_HomingActionType.Dog_Detection;
        stAdvHomePara_Set.stHomingCommand[0].bSlowVelo := FALSE;
        stAdvHomePara_Set.stHomingCommand[0].stStepFuncParameter.eHome_Direction := MC_Home_Direction.mcPositiveDirection;
        stAdvHomePara_Set.stHomingCommand[0].stStepFuncParameter.eSwitch_Mode := MC_Switch_Mode.mcOn;

        //Escape from Home and Re-Enter
        stAdvHomePara_Set.stHomingCommand[1].eHome_ActionType := E_HomingActionType.Dog_Detection;
        stAdvHomePara_Set.stHomingCommand[1].bSlowVelo := TRUE;
        stAdvHomePara_Set.stHomingCommand[1].stStepFuncParameter.eHome_Direction := MC_Home_Direction.mcSwitchNegative;
        stAdvHomePara_Set.stHomingCommand[1].stStepFuncParameter.eSwitch_Mode := MC_Switch_Mode.mcRisingEdge;

        //Neg Find Pulse
        stAdvHomePara_Set.stHomingCommand[2].eHome_ActionType := E_HomingActionType.Index_Detection;
        stAdvHomePara_Set.stHomingCommand[2].bSlowVelo := TRUE;
        stAdvHomePara_Set.stHomingCommand[2].stStepFuncParameter.eHome_Direction := MC_Home_Direction.mcNegativeDirection;

        //Shift Distance
        stAdvHomePara_Set.stHomingCommand[3].eHome_ActionType := E_HomingActionType.FinishHoming;
        stAdvHomePara_Set.stHomingCommand[3].bSlowVelo := TRUE;

        IF NOT bSetPostionBias THEN

            //Set Position
            stAdvHomePara_Set.stHomingCommand[4].eHome_ActionType := E_HomingActionType.HomeDirect;

            stAdvHomePara_Set.uiCommandNum := 5;

        ELSE
            //Set Bias
            stAdvHomePara_Set.stHomingCommand[4].eHome_ActionType := E_HomingActionType.ParameterSetting;

            //Set Position
            stAdvHomePara_Set.stHomingCommand[5].eHome_ActionType := E_HomingActionType.HomeDirect;

            stAdvHomePara_Set.uiCommandNum := 6;
        END_IF

    E_HomingMode._10_Pos_HomeOutterRightIndex_withLimit: //Done

        //Find Home +
        stAdvHomePara_Set.stHomingCommand[0].eHome_ActionType := E_HomingActionType.Dog_Detection;
        stAdvHomePara_Set.stHomingCommand[0].bSlowVelo := FALSE;
        stAdvHomePara_Set.stHomingCommand[0].stStepFuncParameter.eHome_Direction := MC_Home_Direction.mcPositiveDirection;
        stAdvHomePara_Set.stHomingCommand[0].stStepFuncParameter.eSwitch_Mode := MC_Switch_Mode.mcOn;

        //Pos Escape from Home
        stAdvHomePara_Set.stHomingCommand[1].eHome_ActionType := E_HomingActionType.Dog_Detection;
        stAdvHomePara_Set.stHomingCommand[1].bSlowVelo := TRUE;
        stAdvHomePara_Set.stHomingCommand[1].stStepFuncParameter.eHome_Direction := MC_Home_Direction.mcPositiveDirection;
        stAdvHomePara_Set.stHomingCommand[1].stStepFuncParameter.eSwitch_Mode := MC_Switch_Mode.mcFallingEdge;

        //Pos Find Pulse
        stAdvHomePara_Set.stHomingCommand[2].eHome_ActionType := E_HomingActionType.Index_Detection;
        stAdvHomePara_Set.stHomingCommand[2].bSlowVelo := TRUE;
        stAdvHomePara_Set.stHomingCommand[2].stStepFuncParameter.eHome_Direction := MC_Home_Direction.mcPositiveDirection;

        //Shift Distance
        stAdvHomePara_Set.stHomingCommand[3].eHome_ActionType := E_HomingActionType.FinishHoming;
        stAdvHomePara_Set.stHomingCommand[3].bSlowVelo := TRUE;

        IF NOT bSetPostionBias THEN

            //Set Position
            stAdvHomePara_Set.stHomingCommand[4].eHome_ActionType := E_HomingActionType.HomeDirect;

            stAdvHomePara_Set.uiCommandNum := 5;

        ELSE
            //Set Bias
            stAdvHomePara_Set.stHomingCommand[4].eHome_ActionType := E_HomingActionType.ParameterSetting;

            //Set Position
            stAdvHomePara_Set.stHomingCommand[5].eHome_ActionType := E_HomingActionType.HomeDirect;

            stAdvHomePara_Set.uiCommandNum := 6;
        END_IF

    E_HomingMode._11_Neg_HomeOutterRightIndex_withLimit: //Done

        //Find Home -
        stAdvHomePara_Set.stHomingCommand[0].eHome_ActionType := E_HomingActionType.Dog_Detection;
        stAdvHomePara_Set.stHomingCommand[0].bSlowVelo := FALSE;
        stAdvHomePara_Set.stHomingCommand[0].stStepFuncParameter.eHome_Direction := MC_Home_Direction.mcNegativeDirection;
        stAdvHomePara_Set.stHomingCommand[0].stStepFuncParameter.eSwitch_Mode := MC_Switch_Mode.mcOn;

        //Pos Escape from Home
        stAdvHomePara_Set.stHomingCommand[1].eHome_ActionType := E_HomingActionType.Dog_Detection;
        stAdvHomePara_Set.stHomingCommand[1].bSlowVelo := TRUE;
        stAdvHomePara_Set.stHomingCommand[1].stStepFuncParameter.eHome_Direction := MC_Home_Direction.mcPositiveDirection;
        stAdvHomePara_Set.stHomingCommand[1].stStepFuncParameter.eSwitch_Mode := MC_Switch_Mode.mcFallingEdge;

        //Pos Find Pulse
        stAdvHomePara_Set.stHomingCommand[2].eHome_ActionType := E_HomingActionType.Index_Detection;
        stAdvHomePara_Set.stHomingCommand[2].bSlowVelo := TRUE;
        stAdvHomePara_Set.stHomingCommand[2].stStepFuncParameter.eHome_Direction := MC_Home_Direction.mcPositiveDirection;

        //Shift Distance
        stAdvHomePara_Set.stHomingCommand[3].eHome_ActionType := E_HomingActionType.FinishHoming;
        stAdvHomePara_Set.stHomingCommand[3].bSlowVelo := TRUE;

        IF NOT bSetPostionBias THEN

            //Set Position
            stAdvHomePara_Set.stHomingCommand[4].eHome_ActionType := E_HomingActionType.HomeDirect;

            stAdvHomePara_Set.uiCommandNum := 5;

        ELSE
            //Set Bias
            stAdvHomePara_Set.stHomingCommand[4].eHome_ActionType := E_HomingActionType.ParameterSetting;

            //Set Position
            stAdvHomePara_Set.stHomingCommand[5].eHome_ActionType := E_HomingActionType.HomeDirect;

            stAdvHomePara_Set.uiCommandNum := 6;
        END_IF

    E_HomingMode._12_Neg_HomeInnerRightIndex_withLimit:

        //Find Home -
        stAdvHomePara_Set.stHomingCommand[0].eHome_ActionType := E_HomingActionType.Dog_Detection;
        stAdvHomePara_Set.stHomingCommand[0].bSlowVelo := FALSE;
        stAdvHomePara_Set.stHomingCommand[0].stStepFuncParameter.eHome_Direction :=
            MC_Home_Direction.mcNegativeDirection; //MC_Home_Direction.mcSwitchNegative;

        stAdvHomePara_Set.stHomingCommand[0].stStepFuncParameter.eSwitch_Mode := MC_Switch_Mode.mcOn; //MC_Switch_Mode.mcEdgeSwitchNegative;

        //Escape from Home and Re-Enter
        stAdvHomePara_Set.stHomingCommand[1].eHome_ActionType := E_HomingActionType.Dog_Detection;
        stAdvHomePara_Set.stHomingCommand[1].bSlowVelo := TRUE;
        stAdvHomePara_Set.stHomingCommand[1].stStepFuncParameter.eHome_Direction := MC_Home_Direction.mcSwitchNegative;
        stAdvHomePara_Set.stHomingCommand[1].stStepFuncParameter.eSwitch_Mode := MC_Switch_Mode.mcRisingEdge;

        //Neg Find Pulse
        stAdvHomePara_Set.stHomingCommand[2].eHome_ActionType := E_HomingActionType.Index_Detection;
        stAdvHomePara_Set.stHomingCommand[2].bSlowVelo := TRUE;
        stAdvHomePara_Set.stHomingCommand[2].stStepFuncParameter.eHome_Direction := MC_Home_Direction.mcNegativeDirection;

        //Shift Distance
        stAdvHomePara_Set.stHomingCommand[3].eHome_ActionType := E_HomingActionType.FinishHoming;
        stAdvHomePara_Set.stHomingCommand[3].bSlowVelo := TRUE;

        IF NOT bSetPostionBias THEN

            //Set Position
            stAdvHomePara_Set.stHomingCommand[4].eHome_ActionType := E_HomingActionType.HomeDirect;

            stAdvHomePara_Set.uiCommandNum := 5;

        ELSE
            //Set Bias
            stAdvHomePara_Set.stHomingCommand[4].eHome_ActionType := E_HomingActionType.ParameterSetting;

            //Set Position
            stAdvHomePara_Set.stHomingCommand[5].eHome_ActionType := E_HomingActionType.HomeDirect;

            stAdvHomePara_Set.uiCommandNum := 6;
        END_IF

    E_HomingMode._13_Neg_HomeInnerLeftIndex_withLimit:

        //Find Home -
        stAdvHomePara_Set.stHomingCommand[0].eHome_ActionType := E_HomingActionType.Dog_Detection;
        stAdvHomePara_Set.stHomingCommand[0].bSlowVelo := FALSE;
        stAdvHomePara_Set.stHomingCommand[0].stStepFuncParameter.eHome_Direction := MC_Home_Direction.mcNegativeDirection;
        stAdvHomePara_Set.stHomingCommand[0].stStepFuncParameter.eSwitch_Mode := MC_Switch_Mode.mcOn;

        //Neg Escape from Home
        stAdvHomePara_Set.stHomingCommand[1].eHome_ActionType := E_HomingActionType.Dog_Detection;
        stAdvHomePara_Set.stHomingCommand[1].bSlowVelo := TRUE;
        stAdvHomePara_Set.stHomingCommand[1].stStepFuncParameter.eHome_Direction := MC_Home_Direction.mcNegativeDirection;
        stAdvHomePara_Set.stHomingCommand[1].stStepFuncParameter.eSwitch_Mode := MC_Switch_Mode.mcFallingEdge;

        //Find Home +
        stAdvHomePara_Set.stHomingCommand[2].eHome_ActionType := E_HomingActionType.Dog_Detection;
        stAdvHomePara_Set.stHomingCommand[2].bSlowVelo := TRUE;
        stAdvHomePara_Set.stHomingCommand[2].stStepFuncParameter.eHome_Direction := MC_Home_Direction.mcPositiveDirection;
        stAdvHomePara_Set.stHomingCommand[2].stStepFuncParameter.eSwitch_Mode := MC_Switch_Mode.mcRisingEdge;

        //Pos Find Pulse
        stAdvHomePara_Set.stHomingCommand[3].eHome_ActionType := E_HomingActionType.Index_Detection;
        stAdvHomePara_Set.stHomingCommand[3].bSlowVelo := TRUE;
        stAdvHomePara_Set.stHomingCommand[3].stStepFuncParameter.eHome_Direction := MC_Home_Direction.mcPositiveDirection;

        //Shift Distance
        stAdvHomePara_Set.stHomingCommand[4].eHome_ActionType := E_HomingActionType.FinishHoming;
        stAdvHomePara_Set.stHomingCommand[4].bSlowVelo := TRUE;

        IF NOT bSetPostionBias THEN

            //Set Position
            stAdvHomePara_Set.stHomingCommand[5].eHome_ActionType := E_HomingActionType.HomeDirect;

            stAdvHomePara_Set.uiCommandNum := 6;

        ELSE
            //Set Bias
            stAdvHomePara_Set.stHomingCommand[5].eHome_ActionType := E_HomingActionType.ParameterSetting;

            //Set Position
            stAdvHomePara_Set.stHomingCommand[6].eHome_ActionType := E_HomingActionType.HomeDirect;

            stAdvHomePara_Set.uiCommandNum := 7;
        END_IF

    E_HomingMode._14_Neg_HomeOutterLeftIndex_withLimit:

        //Find Home -
        stAdvHomePara_Set.stHomingCommand[0].eHome_ActionType := E_HomingActionType.Dog_Detection;
        stAdvHomePara_Set.stHomingCommand[0].bSlowVelo := FALSE;
        stAdvHomePara_Set.stHomingCommand[0].stStepFuncParameter.eHome_Direction := MC_Home_Direction.mcNegativeDirection;
        stAdvHomePara_Set.stHomingCommand[0].stStepFuncParameter.eSwitch_Mode := MC_Switch_Mode.mcOn;

        //Neg Escape from Home
        stAdvHomePara_Set.stHomingCommand[1].eHome_ActionType := E_HomingActionType.Dog_Detection;
        stAdvHomePara_Set.stHomingCommand[1].bSlowVelo := TRUE;
        stAdvHomePara_Set.stHomingCommand[1].stStepFuncParameter.eHome_Direction := MC_Home_Direction.mcNegativeDirection;
        stAdvHomePara_Set.stHomingCommand[1].stStepFuncParameter.eSwitch_Mode := MC_Switch_Mode.mcFallingEdge;

        //Neg Find Pulse
        stAdvHomePara_Set.stHomingCommand[2].eHome_ActionType := E_HomingActionType.Index_Detection;
        stAdvHomePara_Set.stHomingCommand[2].bSlowVelo := TRUE;
        stAdvHomePara_Set.stHomingCommand[2].stStepFuncParameter.eHome_Direction := MC_Home_Direction.mcNegativeDirection;

        //Shift Distance
        stAdvHomePara_Set.stHomingCommand[3].eHome_ActionType := E_HomingActionType.FinishHoming;
        stAdvHomePara_Set.stHomingCommand[3].bSlowVelo := TRUE;

        IF NOT bSetPostionBias THEN

            //Set Position
            stAdvHomePara_Set.stHomingCommand[4].eHome_ActionType := E_HomingActionType.HomeDirect;

            stAdvHomePara_Set.uiCommandNum := 5;

        ELSE
            //Set Bias
            stAdvHomePara_Set.stHomingCommand[4].eHome_ActionType := E_HomingActionType.ParameterSetting;

            //Set Position
            stAdvHomePara_Set.stHomingCommand[5].eHome_ActionType := E_HomingActionType.HomeDirect;

            stAdvHomePara_Set.uiCommandNum := 6;
        END_IF

    (*-----------------------------------*)
    E_HomingMode._17_Neg_LimitOutterRight:

        //Ref Limit Siganl
        stAdvHomePara_Set.bRefNegLimitSignal := TRUE;

        //Find Limit -
        stAdvHomePara_Set.stHomingCommand[0].eHome_ActionType := E_HomingActionType.Limit_Detection;
        stAdvHomePara_Set.stHomingCommand[0].bSlowVelo := FALSE;
        stAdvHomePara_Set.stHomingCommand[0].stStepFuncParameter.eHome_Direction := MC_Home_Direction.mcNegativeDirection;
        stAdvHomePara_Set.stHomingCommand[0].stStepFuncParameter.eSwitch_Mode := MC_Switch_Mode.mcOn;

        //Escape from Limit
        stAdvHomePara_Set.stHomingCommand[1].eHome_ActionType := E_HomingActionType.Limit_Detection;
        stAdvHomePara_Set.stHomingCommand[1].bSlowVelo := TRUE;
        stAdvHomePara_Set.stHomingCommand[1].stStepFuncParameter.eHome_Direction := MC_Home_Direction.mcNegativeDirection;
        stAdvHomePara_Set.stHomingCommand[1].stStepFuncParameter.eSwitch_Mode := MC_Switch_Mode.mcFallingEdge;

        //Shift Distance
        stAdvHomePara_Set.stHomingCommand[2].eHome_ActionType := E_HomingActionType.FinishHoming;
        stAdvHomePara_Set.stHomingCommand[2].bSlowVelo := TRUE;

        IF NOT bSetPostionBias THEN

            //Set Position
            stAdvHomePara_Set.stHomingCommand[3].eHome_ActionType := E_HomingActionType.HomeDirect;

            stAdvHomePara_Set.uiCommandNum := 4;

        ELSE
            //Set Bias
            stAdvHomePara_Set.stHomingCommand[3].eHome_ActionType := E_HomingActionType.ParameterSetting;

            //Set Position
            stAdvHomePara_Set.stHomingCommand[4].eHome_ActionType := E_HomingActionType.HomeDirect;

            stAdvHomePara_Set.uiCommandNum := 5;
        END_IF

    E_HomingMode._18_Pos_LimitOutterLeft:

        //Ref Limit Siganl
        stAdvHomePara_Set.bRefNegLimitSignal := FALSE;

        //Find Limit +
        stAdvHomePara_Set.stHomingCommand[0].eHome_ActionType := E_HomingActionType.Limit_Detection;
        stAdvHomePara_Set.stHomingCommand[0].bSlowVelo := FALSE;
        stAdvHomePara_Set.stHomingCommand[0].stStepFuncParameter.eHome_Direction := MC_Home_Direction.mcPositiveDirection;
        stAdvHomePara_Set.stHomingCommand[0].stStepFuncParameter.eSwitch_Mode := MC_Switch_Mode.mcOn;

        //Escape from Limit
        stAdvHomePara_Set.stHomingCommand[1].eHome_ActionType := E_HomingActionType.Limit_Detection;
        stAdvHomePara_Set.stHomingCommand[1].bSlowVelo := TRUE;
        stAdvHomePara_Set.stHomingCommand[1].stStepFuncParameter.eHome_Direction := MC_Home_Direction.mcPositiveDirection;
        stAdvHomePara_Set.stHomingCommand[1].stStepFuncParameter.eSwitch_Mode := MC_Switch_Mode.mcFallingEdge;

        //Shift Distance
        stAdvHomePara_Set.stHomingCommand[2].eHome_ActionType := E_HomingActionType.FinishHoming;
        stAdvHomePara_Set.stHomingCommand[2].bSlowVelo := TRUE;

        IF NOT bSetPostionBias THEN

            //Set Position
            stAdvHomePara_Set.stHomingCommand[3].eHome_ActionType := E_HomingActionType.HomeDirect;

            stAdvHomePara_Set.uiCommandNum := 4;

        ELSE
            //Set Bias
            stAdvHomePara_Set.stHomingCommand[3].eHome_ActionType := E_HomingActionType.ParameterSetting;

            //Set Position
            stAdvHomePara_Set.stHomingCommand[4].eHome_ActionType := E_HomingActionType.HomeDirect;

            stAdvHomePara_Set.uiCommandNum := 5;
        END_IF

    E_HomingMode._19_Pos_HomeOutterLeft:

        //Find Home +
        stAdvHomePara_Set.stHomingCommand[0].eHome_ActionType := E_HomingActionType.Dog_Detection;
        stAdvHomePara_Set.stHomingCommand[0].bSlowVelo := FALSE;
        stAdvHomePara_Set.stHomingCommand[0].stStepFuncParameter.eHome_Direction := MC_Home_Direction.mcPositiveDirection;
        stAdvHomePara_Set.stHomingCommand[0].stStepFuncParameter.eSwitch_Mode := MC_Switch_Mode.mcOn;

        //Neg Escpape From Home
        stAdvHomePara_Set.stHomingCommand[1].eHome_ActionType := E_HomingActionType.Dog_Detection;
        stAdvHomePara_Set.stHomingCommand[1].bSlowVelo := TRUE;
        stAdvHomePara_Set.stHomingCommand[1].stStepFuncParameter.eHome_Direction := MC_Home_Direction.mcNegativeDirection;
        stAdvHomePara_Set.stHomingCommand[1].stStepFuncParameter.eSwitch_Mode := MC_Switch_Mode.mcFallingEdge;

        //Shift Distance
        stAdvHomePara_Set.stHomingCommand[2].eHome_ActionType := E_HomingActionType.FinishHoming;
        stAdvHomePara_Set.stHomingCommand[2].bSlowVelo := TRUE;

        IF NOT bSetPostionBias THEN

            //Set Position
            stAdvHomePara_Set.stHomingCommand[3].eHome_ActionType := E_HomingActionType.HomeDirect;

            stAdvHomePara_Set.uiCommandNum := 4;

        ELSE
            //Set Bias
            stAdvHomePara_Set.stHomingCommand[3].eHome_ActionType := E_HomingActionType.ParameterSetting;

            //Set Position
            stAdvHomePara_Set.stHomingCommand[4].eHome_ActionType := E_HomingActionType.HomeDirect;

            stAdvHomePara_Set.uiCommandNum := 5;
        END_IF

    E_HomingMode._20_Pos_HomeInnerLeft:

        //Find Home +
        stAdvHomePara_Set.stHomingCommand[0].eHome_ActionType := E_HomingActionType.Dog_Detection;
        stAdvHomePara_Set.stHomingCommand[0].bSlowVelo := FALSE;
        stAdvHomePara_Set.stHomingCommand[0].stStepFuncParameter.eHome_Direction := MC_Home_Direction.mcPositiveDirection;
        stAdvHomePara_Set.stHomingCommand[0].stStepFuncParameter.eSwitch_Mode := MC_Switch_Mode.mcOn;

        //Escape from Home and Re-Enter
        stAdvHomePara_Set.stHomingCommand[1].eHome_ActionType := E_HomingActionType.Dog_Detection;
        stAdvHomePara_Set.stHomingCommand[1].bSlowVelo := TRUE;
        stAdvHomePara_Set.stHomingCommand[1].stStepFuncParameter.eHome_Direction := MC_Home_Direction.mcSwitchPositive;
        stAdvHomePara_Set.stHomingCommand[1].stStepFuncParameter.eSwitch_Mode := MC_Switch_Mode.mcRisingEdge;

        //Shift Distance
        stAdvHomePara_Set.stHomingCommand[2].eHome_ActionType := E_HomingActionType.FinishHoming;
        stAdvHomePara_Set.stHomingCommand[2].bSlowVelo := TRUE;

        IF NOT bSetPostionBias THEN

            //Set Position
            stAdvHomePara_Set.stHomingCommand[3].eHome_ActionType := E_HomingActionType.HomeDirect;

            stAdvHomePara_Set.uiCommandNum := 4;

        ELSE
            //Set Bias
            stAdvHomePara_Set.stHomingCommand[3].eHome_ActionType := E_HomingActionType.ParameterSetting;

            //Set Position
            stAdvHomePara_Set.stHomingCommand[4].eHome_ActionType := E_HomingActionType.HomeDirect;

            stAdvHomePara_Set.uiCommandNum := 5;
        END_IF

    E_HomingMode._21_Neg_HomeOutterRight:

        //Find Home -
        stAdvHomePara_Set.stHomingCommand[0].eHome_ActionType := E_HomingActionType.Dog_Detection;
        stAdvHomePara_Set.stHomingCommand[0].bSlowVelo := FALSE;
        stAdvHomePara_Set.stHomingCommand[0].stStepFuncParameter.eHome_Direction := MC_Home_Direction.mcNegativeDirection;
        stAdvHomePara_Set.stHomingCommand[0].stStepFuncParameter.eSwitch_Mode := MC_Switch_Mode.mcOn;

        //Escape from Limit 
        stAdvHomePara_Set.stHomingCommand[1].eHome_ActionType := E_HomingActionType.Dog_Detection;
        stAdvHomePara_Set.stHomingCommand[1].bSlowVelo := TRUE;
        stAdvHomePara_Set.stHomingCommand[1].stStepFuncParameter.eHome_Direction := MC_Home_Direction.mcPositiveDirection;
        stAdvHomePara_Set.stHomingCommand[1].stStepFuncParameter.eSwitch_Mode := MC_Switch_Mode.mcFallingEdge;

        //Shift Distance
        stAdvHomePara_Set.stHomingCommand[2].eHome_ActionType := E_HomingActionType.FinishHoming;
        stAdvHomePara_Set.stHomingCommand[2].bSlowVelo := TRUE;

        IF NOT bSetPostionBias THEN

            //Set Position
            stAdvHomePara_Set.stHomingCommand[3].eHome_ActionType := E_HomingActionType.HomeDirect;

            stAdvHomePara_Set.uiCommandNum := 4;

        ELSE
            //Set Bias
            stAdvHomePara_Set.stHomingCommand[3].eHome_ActionType := E_HomingActionType.ParameterSetting;

            //Set Position
            stAdvHomePara_Set.stHomingCommand[4].eHome_ActionType := E_HomingActionType.HomeDirect;

            stAdvHomePara_Set.uiCommandNum := 5;
        END_IF

    E_HomingMode._22_Neg_HomeInnerRight:

        //Find Home -
        stAdvHomePara_Set.stHomingCommand[0].eHome_ActionType := E_HomingActionType.Dog_Detection;
        stAdvHomePara_Set.stHomingCommand[0].bSlowVelo := FALSE;
        stAdvHomePara_Set.stHomingCommand[0].stStepFuncParameter.eHome_Direction := MC_Home_Direction.mcSwitchNegative;
        stAdvHomePara_Set.stHomingCommand[0].stStepFuncParameter.eSwitch_Mode := MC_Switch_Mode.mcOn;

        //Escape from Home and Re-Enter
        stAdvHomePara_Set.stHomingCommand[1].eHome_ActionType := E_HomingActionType.Dog_Detection;
        stAdvHomePara_Set.stHomingCommand[1].bSlowVelo := TRUE;
        stAdvHomePara_Set.stHomingCommand[1].stStepFuncParameter.eHome_Direction := MC_Home_Direction.mcSwitchNegative;
        stAdvHomePara_Set.stHomingCommand[1].stStepFuncParameter.eSwitch_Mode := MC_Switch_Mode.mcRisingEdge;

        //Shift Distance
        stAdvHomePara_Set.stHomingCommand[2].eHome_ActionType := E_HomingActionType.FinishHoming;
        stAdvHomePara_Set.stHomingCommand[2].bSlowVelo := TRUE;

        IF NOT bSetPostionBias THEN

            //Set Position
            stAdvHomePara_Set.stHomingCommand[3].eHome_ActionType := E_HomingActionType.HomeDirect;

            stAdvHomePara_Set.uiCommandNum := 4;

        ELSE
            //Set Bias
            stAdvHomePara_Set.stHomingCommand[3].eHome_ActionType := E_HomingActionType.ParameterSetting;

            //Set Position
            stAdvHomePara_Set.stHomingCommand[4].eHome_ActionType := E_HomingActionType.HomeDirect;

            stAdvHomePara_Set.uiCommandNum := 5;
        END_IF

    E_HomingMode._23_Pos_HomeOutterLeft_withLimit:

        //Pos Find Home
        stAdvHomePara_Set.stHomingCommand[0].eHome_ActionType := E_HomingActionType.Dog_Detection;
        stAdvHomePara_Set.stHomingCommand[0].bSlowVelo := FALSE;
        stAdvHomePara_Set.stHomingCommand[0].stStepFuncParameter.eHome_Direction := MC_Home_Direction.mcPositiveDirection;
        stAdvHomePara_Set.stHomingCommand[0].stStepFuncParameter.eSwitch_Mode := MC_Switch_Mode.mcOn;

        //Neg Escape from Home
        stAdvHomePara_Set.stHomingCommand[1].eHome_ActionType := E_HomingActionType.Dog_Detection;
        stAdvHomePara_Set.stHomingCommand[1].bSlowVelo := TRUE;
        stAdvHomePara_Set.stHomingCommand[1].stStepFuncParameter.eHome_Direction := MC_Home_Direction.mcNegativeDirection;
        stAdvHomePara_Set.stHomingCommand[1].stStepFuncParameter.eSwitch_Mode := MC_Switch_Mode.mcFallingEdge;

        //Shift Distance
        stAdvHomePara_Set.stHomingCommand[2].eHome_ActionType := E_HomingActionType.FinishHoming;
        stAdvHomePara_Set.stHomingCommand[2].bSlowVelo := TRUE;

        IF NOT bSetPostionBias THEN

            //Set Position
            stAdvHomePara_Set.stHomingCommand[3].eHome_ActionType := E_HomingActionType.HomeDirect;

            stAdvHomePara_Set.uiCommandNum := 4;

        ELSE
            //Set Bias
            stAdvHomePara_Set.stHomingCommand[3].eHome_ActionType := E_HomingActionType.ParameterSetting;

            //Set Position
            stAdvHomePara_Set.stHomingCommand[4].eHome_ActionType := E_HomingActionType.HomeDirect;

            stAdvHomePara_Set.uiCommandNum := 5;
        END_IF

    E_HomingMode._24_Pos_HomeInnerLeft_withLimit:

        //Find Home +
        stAdvHomePara_Set.stHomingCommand[0].eHome_ActionType := E_HomingActionType.Dog_Detection;
        stAdvHomePara_Set.stHomingCommand[0].bSlowVelo := FALSE;
        stAdvHomePara_Set.stHomingCommand[0].stStepFuncParameter.eHome_Direction := MC_Home_Direction.mcPositiveDirection;
        stAdvHomePara_Set.stHomingCommand[0].stStepFuncParameter.eSwitch_Mode := MC_Switch_Mode.mcOn;

        //Escape from Home and Re-Enter
        stAdvHomePara_Set.stHomingCommand[1].eHome_ActionType := E_HomingActionType.Dog_Detection;
        stAdvHomePara_Set.stHomingCommand[1].bSlowVelo := TRUE;
        stAdvHomePara_Set.stHomingCommand[1].stStepFuncParameter.eHome_Direction := MC_Home_Direction.mcSwitchPositive;
        stAdvHomePara_Set.stHomingCommand[1].stStepFuncParameter.eSwitch_Mode := MC_Switch_Mode.mcRisingEdge;

        //Shift Distance
        stAdvHomePara_Set.stHomingCommand[2].eHome_ActionType := E_HomingActionType.FinishHoming;
        stAdvHomePara_Set.stHomingCommand[2].bSlowVelo := TRUE;

        IF NOT bSetPostionBias THEN

            //Set Position
            stAdvHomePara_Set.stHomingCommand[3].eHome_ActionType := E_HomingActionType.HomeDirect;

            stAdvHomePara_Set.uiCommandNum := 4;

        ELSE
            //Set Bias
            stAdvHomePara_Set.stHomingCommand[3].eHome_ActionType := E_HomingActionType.ParameterSetting;

            //Set Position
            stAdvHomePara_Set.stHomingCommand[4].eHome_ActionType := E_HomingActionType.HomeDirect;

            stAdvHomePara_Set.uiCommandNum := 5;
        END_IF

    E_HomingMode._25_Pos_HomeInnerRight_withLimit:

        //Find Home +
        stAdvHomePara_Set.stHomingCommand[0].eHome_ActionType := E_HomingActionType.Dog_Detection;
        stAdvHomePara_Set.stHomingCommand[0].bSlowVelo := FALSE;
        stAdvHomePara_Set.stHomingCommand[0].stStepFuncParameter.eHome_Direction := MC_Home_Direction.mcPositiveDirection;
        stAdvHomePara_Set.stHomingCommand[0].stStepFuncParameter.eSwitch_Mode := MC_Switch_Mode.mcOn;

        //Escape from Home and Re-Enter
        stAdvHomePara_Set.stHomingCommand[1].eHome_ActionType := E_HomingActionType.Dog_Detection;
        stAdvHomePara_Set.stHomingCommand[1].bSlowVelo := TRUE;
        stAdvHomePara_Set.stHomingCommand[1].stStepFuncParameter.eHome_Direction := MC_Home_Direction.mcSwitchNegative;
        stAdvHomePara_Set.stHomingCommand[1].stStepFuncParameter.eSwitch_Mode := MC_Switch_Mode.mcRisingEdge;

        //Shift Distance
        stAdvHomePara_Set.stHomingCommand[2].eHome_ActionType := E_HomingActionType.FinishHoming;
        stAdvHomePara_Set.stHomingCommand[2].bSlowVelo := TRUE;

        IF NOT bSetPostionBias THEN

            //Set Position
            stAdvHomePara_Set.stHomingCommand[3].eHome_ActionType := E_HomingActionType.HomeDirect;

            stAdvHomePara_Set.uiCommandNum := 4;

        ELSE
            //Set Bias
            stAdvHomePara_Set.stHomingCommand[3].eHome_ActionType := E_HomingActionType.ParameterSetting;

            //Set Position
            stAdvHomePara_Set.stHomingCommand[4].eHome_ActionType := E_HomingActionType.HomeDirect;

            stAdvHomePara_Set.uiCommandNum := 5;
        END_IF

    E_HomingMode._26_Pos_HomeOutterRight_withLimit:

        //Find Home +
        stAdvHomePara_Set.stHomingCommand[0].eHome_ActionType := E_HomingActionType.Dog_Detection;
        stAdvHomePara_Set.stHomingCommand[0].bSlowVelo := FALSE;
        stAdvHomePara_Set.stHomingCommand[0].stStepFuncParameter.eHome_Direction := MC_Home_Direction.mcPositiveDirection;
        stAdvHomePara_Set.stHomingCommand[0].stStepFuncParameter.eSwitch_Mode := MC_Switch_Mode.mcOn;

        //Pos Escape from Home
        stAdvHomePara_Set.stHomingCommand[1].eHome_ActionType := E_HomingActionType.Dog_Detection;
        stAdvHomePara_Set.stHomingCommand[1].bSlowVelo := TRUE;
        stAdvHomePara_Set.stHomingCommand[1].stStepFuncParameter.eHome_Direction := MC_Home_Direction.mcPositiveDirection;
        stAdvHomePara_Set.stHomingCommand[1].stStepFuncParameter.eSwitch_Mode := MC_Switch_Mode.mcFallingEdge;

        //Shift Distance
        stAdvHomePara_Set.stHomingCommand[2].eHome_ActionType := E_HomingActionType.FinishHoming;
        stAdvHomePara_Set.stHomingCommand[2].bSlowVelo := TRUE;

        IF NOT bSetPostionBias THEN

            //Set Position
            stAdvHomePara_Set.stHomingCommand[3].eHome_ActionType := E_HomingActionType.HomeDirect;

            stAdvHomePara_Set.uiCommandNum := 4;

        ELSE
            //Set Bias
            stAdvHomePara_Set.stHomingCommand[3].eHome_ActionType := E_HomingActionType.ParameterSetting;

            //Set Position
            stAdvHomePara_Set.stHomingCommand[4].eHome_ActionType := E_HomingActionType.HomeDirect;

            stAdvHomePara_Set.uiCommandNum := 5;
        END_IF

    E_HomingMode._27_Neg_HomeOutterRight_withLimit:

        //Find Home -
        stAdvHomePara_Set.stHomingCommand[0].eHome_ActionType := E_HomingActionType.Dog_Detection;
        stAdvHomePara_Set.stHomingCommand[0].bSlowVelo := FALSE;
        stAdvHomePara_Set.stHomingCommand[0].stStepFuncParameter.eHome_Direction := MC_Home_Direction.mcNegativeDirection;
        stAdvHomePara_Set.stHomingCommand[0].stStepFuncParameter.eSwitch_Mode := MC_Switch_Mode.mcOn;

        //Pos Escape from Home
        stAdvHomePara_Set.stHomingCommand[1].eHome_ActionType := E_HomingActionType.Dog_Detection;
        stAdvHomePara_Set.stHomingCommand[1].bSlowVelo := TRUE;
        stAdvHomePara_Set.stHomingCommand[1].stStepFuncParameter.eHome_Direction := MC_Home_Direction.mcPositiveDirection;
        stAdvHomePara_Set.stHomingCommand[1].stStepFuncParameter.eSwitch_Mode := MC_Switch_Mode.mcFallingEdge;

        //Shift Distance
        stAdvHomePara_Set.stHomingCommand[2].eHome_ActionType := E_HomingActionType.FinishHoming;
        stAdvHomePara_Set.stHomingCommand[2].bSlowVelo := TRUE;

        IF NOT bSetPostionBias THEN

            //Set Position
            stAdvHomePara_Set.stHomingCommand[3].eHome_ActionType := E_HomingActionType.HomeDirect;

            stAdvHomePara_Set.uiCommandNum := 4;

        ELSE
            //Set Bias
            stAdvHomePara_Set.stHomingCommand[4].eHome_ActionType := E_HomingActionType.ParameterSetting;

            //Set Position
            stAdvHomePara_Set.stHomingCommand[5].eHome_ActionType := E_HomingActionType.HomeDirect;

            stAdvHomePara_Set.uiCommandNum := 6;
        END_IF

    E_HomingMode._28_Neg_HomeInnerRight_withLimit:

        //Find Home -
        stAdvHomePara_Set.stHomingCommand[0].eHome_ActionType := E_HomingActionType.Dog_Detection;
        stAdvHomePara_Set.stHomingCommand[0].bSlowVelo := FALSE;
        stAdvHomePara_Set.stHomingCommand[0].stStepFuncParameter.eHome_Direction :=
            MC_Home_Direction.mcNegativeDirection; //MC_Home_Direction.mcSwitchNegative;

        stAdvHomePara_Set.stHomingCommand[0].stStepFuncParameter.eSwitch_Mode := MC_Switch_Mode.mcOn; //MC_Switch_Mode.mcEdgeSwitchNegative;

        //Escape from Home and Re-Enter
        stAdvHomePara_Set.stHomingCommand[1].eHome_ActionType := E_HomingActionType.Dog_Detection;
        stAdvHomePara_Set.stHomingCommand[1].bSlowVelo := TRUE;
        stAdvHomePara_Set.stHomingCommand[1].stStepFuncParameter.eHome_Direction := MC_Home_Direction.mcSwitchNegative;
        stAdvHomePara_Set.stHomingCommand[1].stStepFuncParameter.eSwitch_Mode := MC_Switch_Mode.mcRisingEdge;

        //Shift Distance
        stAdvHomePara_Set.stHomingCommand[2].eHome_ActionType := E_HomingActionType.FinishHoming;
        stAdvHomePara_Set.stHomingCommand[2].bSlowVelo := TRUE;

        IF NOT bSetPostionBias THEN

            //Set Position
            stAdvHomePara_Set.stHomingCommand[3].eHome_ActionType := E_HomingActionType.HomeDirect;

            stAdvHomePara_Set.uiCommandNum := 4;
        ELSE
            //Set Bias
            stAdvHomePara_Set.stHomingCommand[3].eHome_ActionType := E_HomingActionType.ParameterSetting;

            //Set Position
            stAdvHomePara_Set.stHomingCommand[4].eHome_ActionType := E_HomingActionType.HomeDirect;

            stAdvHomePara_Set.uiCommandNum := 5;
        END_IF

    E_HomingMode._29_Neg_HomeInnerLeft_withLimit:

        //Find Home -
        stAdvHomePara_Set.stHomingCommand[0].eHome_ActionType := E_HomingActionType.Dog_Detection;
        stAdvHomePara_Set.stHomingCommand[0].bSlowVelo := FALSE;
        stAdvHomePara_Set.stHomingCommand[0].stStepFuncParameter.eHome_Direction := MC_Home_Direction.mcNegativeDirection;
        stAdvHomePara_Set.stHomingCommand[0].stStepFuncParameter.eSwitch_Mode := MC_Switch_Mode.mcOn;

        //Neg Escape from Home
        stAdvHomePara_Set.stHomingCommand[1].eHome_ActionType := E_HomingActionType.Dog_Detection;
        stAdvHomePara_Set.stHomingCommand[1].bSlowVelo := TRUE;
        stAdvHomePara_Set.stHomingCommand[1].stStepFuncParameter.eHome_Direction := MC_Home_Direction.mcNegativeDirection;
        stAdvHomePara_Set.stHomingCommand[1].stStepFuncParameter.eSwitch_Mode := MC_Switch_Mode.mcFallingEdge;

        //Find Home +
        stAdvHomePara_Set.stHomingCommand[2].eHome_ActionType := E_HomingActionType.Dog_Detection;
        stAdvHomePara_Set.stHomingCommand[2].bSlowVelo := TRUE;
        stAdvHomePara_Set.stHomingCommand[2].stStepFuncParameter.eHome_Direction := MC_Home_Direction.mcPositiveDirection;
        stAdvHomePara_Set.stHomingCommand[2].stStepFuncParameter.eSwitch_Mode := MC_Switch_Mode.mcRisingEdge;

        //Shift Distance
        stAdvHomePara_Set.stHomingCommand[3].eHome_ActionType := E_HomingActionType.FinishHoming;
        stAdvHomePara_Set.stHomingCommand[3].bSlowVelo := TRUE;

        IF NOT bSetPostionBias THEN

            //Set Position
            stAdvHomePara_Set.stHomingCommand[4].eHome_ActionType := E_HomingActionType.HomeDirect;

            stAdvHomePara_Set.uiCommandNum := 5;

        ELSE
            //Set Bias
            stAdvHomePara_Set.stHomingCommand[4].eHome_ActionType := E_HomingActionType.ParameterSetting;

            //Set Position
            stAdvHomePara_Set.stHomingCommand[5].eHome_ActionType := E_HomingActionType.HomeDirect;

            stAdvHomePara_Set.uiCommandNum := 6;
        END_IF

    E_HomingMode._30_Neg_HomeOutterLeft_withLimit:

        //Find Home -
        stAdvHomePara_Set.stHomingCommand[0].eHome_ActionType := E_HomingActionType.Dog_Detection;
        stAdvHomePara_Set.stHomingCommand[0].bSlowVelo := FALSE;
        stAdvHomePara_Set.stHomingCommand[0].stStepFuncParameter.eHome_Direction := MC_Home_Direction.mcNegativeDirection;
        stAdvHomePara_Set.stHomingCommand[0].stStepFuncParameter.eSwitch_Mode := MC_Switch_Mode.mcOn;

        //Neg Escape from Home
        stAdvHomePara_Set.stHomingCommand[1].eHome_ActionType := E_HomingActionType.Dog_Detection;
        stAdvHomePara_Set.stHomingCommand[1].bSlowVelo := TRUE;
        stAdvHomePara_Set.stHomingCommand[1].stStepFuncParameter.eHome_Direction := MC_Home_Direction.mcNegativeDirection;
        stAdvHomePara_Set.stHomingCommand[1].stStepFuncParameter.eSwitch_Mode := MC_Switch_Mode.mcFallingEdge;

        //Shift Distance
        stAdvHomePara_Set.stHomingCommand[2].eHome_ActionType := E_HomingActionType.FinishHoming;
        stAdvHomePara_Set.stHomingCommand[2].bSlowVelo := TRUE;

        IF NOT bSetPostionBias THEN

            //Set Position
            stAdvHomePara_Set.stHomingCommand[3].eHome_ActionType := E_HomingActionType.HomeDirect;

            stAdvHomePara_Set.uiCommandNum := 4;

        ELSE
            //Set Bias
            stAdvHomePara_Set.stHomingCommand[3].eHome_ActionType := E_HomingActionType.ParameterSetting;

            //Set Position
            stAdvHomePara_Set.stHomingCommand[4].eHome_ActionType := E_HomingActionType.HomeDirect;

            stAdvHomePara_Set.uiCommandNum := 5;
        END_IF

    E_HomingMode._33_Neg_Index:

        //Neg Find Pulse
        stAdvHomePara_Set.stHomingCommand[0].eHome_ActionType := E_HomingActionType.Index_Detection;
        stAdvHomePara_Set.stHomingCommand[0].bSlowVelo := TRUE;
        stAdvHomePara_Set.stHomingCommand[0].stStepFuncParameter.eHome_Direction := MC_Home_Direction.mcNegativeDirection;

        //Shift Distance
        stAdvHomePara_Set.stHomingCommand[1].eHome_ActionType := E_HomingActionType.FinishHoming;
        stAdvHomePara_Set.stHomingCommand[1].bSlowVelo := TRUE;

        IF NOT bSetPostionBias THEN

            //Set Position
            stAdvHomePara_Set.stHomingCommand[2].eHome_ActionType := E_HomingActionType.HomeDirect;

            stAdvHomePara_Set.uiCommandNum := 3;

        ELSE
            //Set Bias
            stAdvHomePara_Set.stHomingCommand[2].eHome_ActionType := E_HomingActionType.ParameterSetting;

            //Set Position
            stAdvHomePara_Set.stHomingCommand[3].eHome_ActionType := E_HomingActionType.HomeDirect;

            stAdvHomePara_Set.uiCommandNum := 4;
        END_IF

    E_HomingMode._34_Pos_Index: //Done

        //Neg Find Pulse
        stAdvHomePara_Set.stHomingCommand[0].eHome_ActionType := E_HomingActionType.Index_Detection;
        stAdvHomePara_Set.stHomingCommand[0].bSlowVelo := TRUE;
        stAdvHomePara_Set.stHomingCommand[0].stStepFuncParameter.eHome_Direction := MC_Home_Direction.mcPositiveDirection;

        //Shift Distance
        stAdvHomePara_Set.stHomingCommand[1].eHome_ActionType := E_HomingActionType.FinishHoming;
        stAdvHomePara_Set.stHomingCommand[1].bSlowVelo := TRUE;

        IF NOT bSetPostionBias THEN

            //Set Position
            stAdvHomePara_Set.stHomingCommand[2].eHome_ActionType := E_HomingActionType.HomeDirect;

            stAdvHomePara_Set.uiCommandNum := 3;

        ELSE
            //Set Bias
            stAdvHomePara_Set.stHomingCommand[2].eHome_ActionType := E_HomingActionType.ParameterSetting;

            //Set Position
            stAdvHomePara_Set.stHomingCommand[3].eHome_ActionType := E_HomingActionType.HomeDirect;

            stAdvHomePara_Set.uiCommandNum := 4;
        END_IF

    E_HomingMode._35_CurrentPosition:

        IF NOT bSetPostionBias THEN

            //Finish 
            stAdvHomePara_Set.stHomingCommand[0].eHome_ActionType := E_HomingActionType.HomeDirect;

            stAdvHomePara_Set.uiCommandNum := 1;

        ELSE
            //Set Bias
            stAdvHomePara_Set.stHomingCommand[0].eHome_ActionType := E_HomingActionType.ParameterSetting;

            //Finish 
            stAdvHomePara_Set.stHomingCommand[1].eHome_ActionType := E_HomingActionType.HomeDirect;

            stAdvHomePara_Set.uiCommandNum := 2;

        END_IF
	E_HomingMode._36_MoveToAbsHomePoint:
        // Move abs to home point
        stAdvHomePara_Set.stHomingCommand[0].eHome_ActionType := E_HomingActionType.MoveAbs;
        stAdvHomePara_Set.stHomingCommand[0].bSlowVelo := FALSE;

        //Shift Distance
        stAdvHomePara_Set.stHomingCommand[1].eHome_ActionType := E_HomingActionType.FinishHoming;
        stAdvHomePara_Set.stHomingCommand[1].bSlowVelo := TRUE;
		stAdvHomePara_Set.uiCommandNum := 2;
END_CASE
END_METHOD

METHOD M_SetUserDefinedMode : BOOL
VAR_INPUT
END_VAR
END_METHOD

END_FUNCTION_BLOCK

// Basic Function/FB_JsonHandler
FUNCTION_BLOCK FB_JsonHandler EXTENDS FB_ActionBasic
VAR_INPUT
	xExecute	:BOOL;
	
	eAction		: E_JsonHandlerAction;
	sFilePath	: T_MaxString;
	pData		: PVOID;
	nData		: UDINT;
END_VAR
VAR_OUTPUT
	iErrorId	:INT;
END_VAR
VAR
	(* State Machine *)
    StateBehaviour : CBML.ETrig;
	
	//-----FBs-----
	//Json
	fbJsonConverter		:FB_Json_Converter;
	
	//File Handle
	fbFileOpen 	: FB_FileOpen;
	fbFileRead 	: FB_FileRead;
	fbFileWrite : FB_FileWrite;
	fbFileClose : FB_FileClose;
	
	//-----Step-----
	iStep_WriteJson	:INT;
	iStep_ReadJson	:INT;
	
	//-----Var-----
	i						: INT;
	bFileExist				: BOOL;
	sReadFilePath			: T_MaxString;
	sWriteFilePath			: T_MaxString;
	sJsonString_FromFile	: STRING(10000);
	sJsonString_FromObj		: STRING(10000);

	nJsonToObj	:UDINT;
	pJsonToObj	:PVOID;
	nObjToJson	:UDINT;
	pObjToJson	:PVOID;
END_VAR

(* State Machine *)
THIS^.IBehaviourModel := StateBehaviour;
StateBehaviour(xExecute := xExecute, xBusy => xBusy, xDone => xDone, xError => xError);

A_CyclicUpdate();

METHOD CleanupAction
VAR_INPUT
    xAbortProposed : BOOL;
    iErrorIDProposed: INT;
END_VAR
VAR_OUTPUT
    xComplete : BOOL := TRUE;
    xAbort: BOOL := xAbortProposed;
 	iErrorID : INT := iErrorIDProposed;
END_VAR
THIS^.iErrorId := iErrorIDProposed;
END_METHOD

METHOD CyclicAction
VAR_INPUT
    itfTimingController : CBML.ITimingController;
END_VAR
VAR_OUTPUT
    xComplete : BOOL := TRUE;
    iErrorID : INT := 0;
END_VAR
xComplete:=FALSE;
(* ----- Read ----- *)
CASE iStep_ReadJson OF
	1:
		//Reset FBs 
		fbFileOpen.bExecute := FALSE;
		fbFileRead.bExecute := FALSE;
		fbFileWrite.bExecute := FALSE;
		fbFileClose.bExecute := FALSE;
		
		sJsonString_FromFile:='';
		
		iStep_ReadJson:=2;
	2:
		fbFileOpen(
			sPathName:= sReadFilePath,
			nMode:= FOPEN_MODEREAD,
			ePath:= , 
			bExecute:= TRUE);
		
		IF NOT fbFileOpen.bBusy THEN
			
			fbFileOpen.bExecute:=FALSE;
		
			IF fbFileOpen.bError THEN
				
				//Error
				iErrorID := 9900;
				iStep_ReadJson := 99;
				
			ELSE
				IF NOT (fbFileOpen.hFile = 0) THEN
					iStep_ReadJson := 3;
				END_IF
			END_IF
		END_IF
			
	3:
		fbFileRead(
			hFile:= fbFileOpen.hFile, 
			pReadBuff:= ADR(sJsonString_FromFile), 
			cbReadLen:= SIZEOF(sJsonString_FromFile), 
			bExecute:= TRUE);
			
		IF NOT fbFileRead.bBusy THEN
			
			fbFileRead.bExecute:=FALSE;
			
			IF fbFileRead.bError THEN
				
				//Error
				iErrorID := 9901;
				iStep_ReadJson := 99;
				
			ELSE
				iStep_ReadJson := 4;
			END_IF
		END_IF
		
	4:
		//Convert Json string to Object
		fbJsonConverter.JsonStrToObj(JsonStr:= sJsonString_FromFile, nData:= nJsonToObj, pData:= pJsonToObj);
		iStep_ReadJson := 5;
		
	5:
		fbFileClose(
			hFile:= fbFileOpen.hFile, 
			bExecute:= TRUE);
			
		IF NOT fbFileClose.bBusy THEN
			
			fbFileClose.bExecute:=FALSE;
			
			IF fbFileClose.bError THEN
				
				//Error
				iErrorID := 9902;
				
				iStep_ReadJson := 99;
			ELSE
				
				iStep_ReadJson := 10;
			END_IF
		END_IF
	10://Done
		iStep_ReadJson := 0;
		xComplete:=TRUE;
	99://Error
END_CASE


(* ----- Write ----- *)
CASE iStep_WriteJson OF
	1:
		//Reset FBs 
		fbFileOpen.bExecute := FALSE;
		fbFileRead.bExecute := FALSE;
		fbFileWrite.bExecute := FALSE;
		fbFileClose.bExecute := FALSE;
		
		sJsonString_FromObj:='';
		
		iStep_WriteJson:=2;
	2:
		fbFileOpen(
			sPathName:= sWriteFilePath,
			nMode:= FOPEN_MODEWRITE OR FOPEN_MODEPLUS,
			ePath:= , 
			bExecute:= TRUE);
			
		IF NOT fbFileOpen.bBusy THEN
			
			fbFileOpen.bExecute:=FALSE;
			
			IF fbFileOpen.bError THEN
				
				//Error
				iErrorID := 9900;
				
				iStep_WriteJson := 99;
			ELSE
				IF NOT (fbFileOpen.hFile = 0) THEN
					iStep_WriteJson := 3;
				END_IF
			END_IF
		END_IF
		
	3:
		//Convert Object to Json string
		sJsonString_FromObj := fbJsonConverter.ObjToJsonStr(nData:= nObjToJson, pData:= pObjToJson);
		
		iStep_WriteJson := 4;
	4:
		fbFileWrite(
			hFile:= fbFileOpen.hFile, 
			pWriteBuff:= ADR(sJsonString_FromObj), 
			cbWriteLen:= LEN2(ADR(sJsonString_FromObj)),
			bExecute:= TRUE);
			
		IF NOT fbFileWrite.bBusy THEN
			
			fbFileWrite.bExecute:=FALSE;
			
			IF NOT fbFileWrite.bError THEN
				iStep_WriteJson := 5;
			ELSE
				
				//Error
				iErrorID := 9911;
				
				iStep_WriteJson := 99;
			END_IF
		END_IF
			
	5:
		fbFileClose(
			hFile:= fbFileOpen.hFile, 
			bExecute:= TRUE);
		
		IF NOT fbFileClose.bBusy THEN
			fbFileClose.bExecute:=FALSE;
			
			IF NOT fbFileClose.bError THEN
				
				iStep_WriteJson := 10;
			ELSE
				
				//Error
				iErrorID := 9912;
				
				iStep_WriteJson := 99;
			END_IF
		END_IF
			
	10://Done
		xComplete:=TRUE;
		
		iStep_WriteJson:=0;
	99://Error
		//M_SetError(0);
END_CASE
END_METHOD

METHOD StartAction
VAR_OUTPUT
    xComplete : BOOL := TRUE;
	iErrorID : INT := 0;
END_VAR

CASE eAction OF
	
	E_JsonHandlerAction.READ:
	
		nJsonToObj	:= nData;
		pJsonToObj	:= pData;
		
		sReadFilePath := sFilePath;
		
		iStep_ReadJson := 1;
		
	E_JsonHandlerAction.WRITE:
	
		nObjToJson := nData;
		pObjToJson := pData;

		sWriteFilePath := sFilePath;
		
		iStep_WriteJson := 1;
END_CASE
END_METHOD

ACTION A_CyclicUpdate:

//---FB Refresh---
fbJsonConverter();
fbFileOpen();
fbFileRead();
fbFileWrite();
fbFileClose();
END_ACTION

END_FUNCTION_BLOCK

// Basic Function/FB_Json_Converter
FUNCTION_BLOCK FB_Json_Converter
VAR_INPUT
END_VAR
VAR_OUTPUT
END_VAR
VAR
	// json功能块
	fbJsonRWDT 		: FB_JsonReadWriteDataType;
	fbJsonW 		: FB_JsonSaxPrettyWriter;
	fbJsonDP 		: FB_JsonDomParser;
END_VAR

(*
* 功能 1 输入键（字符串）-值（任意数据类型）自动载入json
* 功能 2 输入键（字符串）自动返回值（任意数据类型，包括自定义数据类型以及JSON）
* 功能 3 JSON数据重置
* 功能 4 输出JSON字符串
* 功能 5 输入JSON字符串，转化为Json对象（取消）
* 功能 6 输入特定结构体对象，直接转化为Json字符串并返回
* 功能 7 输入JSON字符串，转化为结构体
*)

METHOD JsonStrToObj : bool
VAR_INPUT
	JsonStr: STRING(100000);
	nData: UDINT;
	pData: PVOID;
END_VAR
VAR
	typestr: STRING;
	hrErrorCode : HRESULT;
END_VAR
(*
* 功能 7 输入JSON字符串，转化为结构体
*)
// 获得值变量的数据类型
typestr := fbJsonRWDT.GetDatatypeNameByAddress(nData := nData, pData := pData);
// 重置Json缓存
fbJsonW.ResetDocument();
// 将JSON字符串的信息写入特定数据
fbJsonRWDT.SetSymbolFromJson(sJson:= JsonStr, sDatatype:= typestr, nData:= nData, pData:= pData,hrErrorCode=>hrErrorCode);
END_METHOD

METHOD ObjToJsonStr : STRING(100000)
VAR_INPUT
	nData: UDINT;
	pData: PVOID;
END_VAR
VAR
	typestr: STRING;
END_VAR
(*
* 功能 6 输入特定结构体对象，直接转化为Json字符串并返回
*)
// 获得值变量的数据类型
typestr := fbJsonRWDT.GetDatatypeNameByAddress(nData := nData, pData := pData);
// 重置Json缓存
fbJsonW.ResetDocument();
//fbJsonW.SetFormatOptions(EJsonPrettyFormatOptions.eFormatSingleLineArray);
// 添加数据到Json缓存
fbJsonRWDT.AddJsonValueFromSymbol(fbJsonW, typestr, nData, pData);

// 将当前缓存转为字符串
fbJsonW.CopyDocument(pDoc:= ObjToJsonStr, nDoc:= SIZEOF(ObjToJsonStr));
END_METHOD

END_FUNCTION_BLOCK

// CorrugatedPrint/Feeder/F_Poly7_MinTime
FUNCTION F_Poly7_MinTime : Lreal
VAR_INPUT
    EndPosition    : LREAL;   // This value is the poly7 end point position [mm]
    EndVelocity    : LREAL;   // This value is the poly7 end point velocity [mm/s]
END_VAR
VAR
    T       : LREAL := 1.0;          // 嘗試時間
    T_step  : LREAL := 0.05;         // 時間步進
    v1      : LREAL;                 // 標準化終點速度
    dy      : LREAL;                 // 導數 dy/dx
    v       : LREAL;                 // 當前速度
    v_peak  : LREAL;                 // 最大速度

    a4, a5, a6, a7 : LREAL;          // Poly7 係數
    ok      : BOOL;                 // 是否成功解係數

    // For 取樣 x
    idx     : INT;
    nSteps  : INT;
    x       : LREAL;
    dx      : LREAL := 0.01;

    i       : INT;
    found   : BOOL := FALSE;
END_VAR

FOR i := 0 TO 380 BY 1 DO // 最多搜尋到 T = 20 秒（(20 - 1) / 0.05 = 380 次）
    T := 0.05 + i * T_step;
    v1 := EndVelocity * T / EndPosition;

    // 解出 Poly7 係數（根據 v1）
    ok := F_SolvePoly7Coefficients(EndVelocity := v1, a4 => a4, a5 => a5, a6 => a6, a7 => a7);

    IF NOT ok THEN
        CONTINUE; // 若解失敗跳過
    END_IF

    // 搜尋 x ∈ [0, 1] 內的速度峰值
    v_peak := 0.0;
    nSteps := LREAL_TO_INT(1.0 / dx);
    FOR idx := 0 TO nSteps DO
        x := idx * dx;
        dy := 4 * a4 * x*x*x + 5 * a5 * x*x*x*x + 6 * a6 * x*x*x*x*x + 7 * a7 * x*x*x*x*x*x;
        v  := EndPosition * dy / T;
        IF v > v_peak THEN
            v_peak := v;
        END_IF
    END_FOR

    // 若整段速度未超過終點速度，視為合法
    IF v_peak <= EndVelocity THEN
        found := TRUE;
        EXIT;
    END_IF
END_FOR

IF found THEN
    F_Poly7_MinTime := T;
ELSE
    F_Poly7_MinTime := -1.0; // 找不到合法時間
END_IF

END_FUNCTION

// CorrugatedPrint/Feeder/F_SolvePoly7Coefficients
FUNCTION F_SolvePoly7Coefficients : bool
VAR_INPUT
    EndVelocity  : LREAL;    // 標準化終點速度 v1 = T * Vend / L
END_VAR
VAR
    A  : ARRAY[1..4, 1..4] OF LREAL;
    b  : ARRAY[1..4] OF LREAL;
    x  : ARRAY[1..4] OF LREAL;
    i, j, k : INT;
    factor, sum : LREAL;
END_VAR
VAR_OUTPUT
    a4  : LREAL;
    a5  : LREAL;
    a6  : LREAL;
    a7  : LREAL;
END_VAR

// 設定係數矩陣 A 與向量 b
A[1,1] := 1;  A[1,2] := 1;  A[1,3] := 1;  A[1,4] := 1;
A[2,1] := 4;  A[2,2] := 5;  A[2,3] := 6;  A[2,4] := 7;
A[3,1] := 12; A[3,2] := 20; A[3,3] := 30; A[3,4] := 42;
A[4,1] := 24; A[4,2] := 60; A[4,3] := 120; A[4,4] := 210;

b[1] := 1.0;
b[2] := EndVelocity;
b[3] := 0.0;
b[4] := 0.0;

// Gaussian Elimination - Forward Elimination
FOR i := 1 TO 3 DO
    FOR j := i + 1 TO 4 DO
        IF A[i,i] = 0 THEN
            F_SolvePoly7Coefficients := FALSE; // Avoid divide by zero
            RETURN;
        END_IF
        factor := A[j,i] / A[i,i];
        FOR k := i TO 4 DO
            A[j,k] := A[j,k] - factor * A[i,k];
        END_FOR
        b[j] := b[j] - factor * b[i];
    END_FOR
END_FOR

// Back Substitution
FOR i := 4 TO 1 BY -1 DO
    sum := 0.0;
    FOR j := i + 1 TO 4 DO
        sum := sum + A[i,j] * x[j];
    END_FOR
    IF A[i,i] = 0 THEN
        F_SolvePoly7Coefficients := FALSE;
        RETURN;
    END_IF
    x[i] := (b[i] - sum) / A[i,i];
END_FOR

// 傳出解
a4 := x[1];
a5 := x[2];
a6 := x[3];
a7 := x[4];

F_SolvePoly7Coefficients := TRUE;

END_FUNCTION

// CorrugatedPrint/Feeder/FB_CorrugatedLiftingCalculate
FUNCTION_BLOCK FB_CorrugatedLiftingCalculate EXTENDS FB_ActionBasic
VAR_INPUT
    xExecute            : BOOL;
    xAbort              : BOOL;
    AxisID              : UDINT; 
    ProfileNum          : UDINT := 1;      // 1~4 

	WorkingAreaStartPos : LREAL; // This value is used to set the working area start position
	WorkingAreaEndPos : LREAL; // This value is used to set the working area end position
    MaxMasterVelocity   : LREAL := 170;    // Machine production per minute. (Sheet/min)
    ProductLength       : LREAL := 1300;   // Corrugate Paper total length
    PrintRollerDiameter : LREAL := 446.17; // PrintRoller Diameter, this value is used to calculate linespeed
	SlaveWorkLength : LREAL;
    WheelThreadPosition : LREAL := 45.8;   // Roller center position (mm)
END_VAR
VAR_OUTPUT
    xAborted : BOOL;
END_VAR
VAR
    StateBehaviour           : CBML.ETrigA;
    arCamPoint               : ARRAY[0..2] OF MC_MotionFunctionPoint;
    PrintCircumference       : LREAL;
    MaxMachineLineSpeed      : LREAL;
    MachineLineSpeed         : LREAL;

    // Calculate Curve
    Curve1_MasterPosition : LREAL; // (deg)
    Curve1_SlavePosition  : LREAL; // (mm)
    Curve2_MasterPosition : LREAL; // (deg)
    Curve2_SlavePosition  : LREAL; // (mm)
    Curve2_SlaveVelocity  : LREAL; // (mm/s)
    Curve3_MasterPosition : LREAL; // (deg)
    Curve3_SlavePosition  : LREAL; // (mm)
END_VAR

THIS^.IBehaviourModel := StateBehaviour;
StateBehaviour(
	xExecute:= xExecute, 
	xDone=> xDone, 
	xBusy=> xBusy, 
	xError=> xError, 
	xAbort:= xAbort,
	xAborted=> xAborted);

METHOD CleanupAction
VAR_INPUT
    xAbortProposed : BOOL;
    iErrorIDProposed: INT;
END_VAR
VAR_OUTPUT
    xComplete : BOOL := TRUE;
    xAbort: BOOL := xAbortProposed;
 	iErrorID : INT := iErrorIDProposed;
END_VAR
END_METHOD

METHOD CyclicAction
VAR_INPUT
    itfTimingController : CBML.ITimingController;
END_VAR
VAR_OUTPUT
    xComplete : BOOL := TRUE;
    iErrorID : INT := 0;
END_VAR

arAxisCtrl_gb[AxisID].SyncMode.SyncProfile.CamProfile[ProfileNum].ArraySize   := SIZEOF(arCamPoint);
arAxisCtrl_gb[AxisID].SyncMode.SyncProfile.CamProfile[ProfileNum].NoOfColumns := 1;
arAxisCtrl_gb[AxisID].SyncMode.SyncProfile.CamProfile[ProfileNum].NoOfRows    := 3;
arAxisCtrl_gb[AxisID].SyncMode.SyncProfile.CamProfile[ProfileNum].pArray      := ADR(arCamPoint);
arAxisCtrl_gb[AxisID].SyncMode.SyncProfile.CamProfile[ProfileNum].TableType   := MC_TABLETYPE_MOTIONFUNCTION;

arCamPoint[0].FunctionType := MOTIONFUNCTYPE_POLYNOM1;
arCamPoint[0].MasterPos    := 0;
arCamPoint[0].SlavePos     := 0;
arCamPoint[0].PointIndex   := 1;
arCamPoint[0].PointType    := MOTIONPOINTTYPE_REST;

arCamPoint[1].FunctionType := MOTIONFUNCTYPE_POLYNOM5;
arCamPoint[1].MasterPos    := Curve1_MasterPosition;
arCamPoint[1].SlavePos     := Curve1_SlavePosition;
arCamPoint[1].PointIndex   := 2;
arCamPoint[1].PointType    := MOTIONPOINTTYPE_REST;

arCamPoint[2].FunctionType := MOTIONFUNCTYPE_POLYNOM5;
arCamPoint[2].MasterPos    := Curve2_MasterPosition;
arCamPoint[2].SlavePos     := Curve2_SlavePosition;
arCamPoint[2].PointIndex   := 3;
arCamPoint[2].PointType    := MOTIONPOINTTYPE_REST;
END_METHOD

METHOD StartAction
VAR_OUTPUT
    xComplete : BOOL := TRUE;
	iErrorID : INT := 0;
END_VAR
// Check Parameter is correct
// Data analyze
PrintCircumference := PrintRollerDiameter * PI; // (mm)
SlaveWorkLength := ProductLength - WheelThreadPosition;

// Data input 
Curve1_MasterPosition := SlaveWorkLength/PrintCircumference *360.0;
Curve1_SlavePosition := 0;
Curve2_MasterPosition := 360.0;
Curve2_SlavePosition := 360;
END_METHOD

END_FUNCTION_BLOCK

// CorrugatedPrint/Feeder/FB_CorrugatedWheelThreadCalculate
FUNCTION_BLOCK FB_CorrugatedWheelThreadCalculate EXTENDS FB_ActionBasic
VAR_INPUT
    xExecute            : BOOL;
    xAbort              : BOOL;
    ProfileNum          : UDINT := 1;      // 1~4 
    MaxMasterVelocity   : LREAL := 170;    // Machine production per minute. (Sheet/min)
    ProductLength       : LREAL := 1300;   // Corrugate Paper total length
    AccDistance         : LREAL := 147.47; // Acceleration distance (mm)
    WheelThreadPosition : LREAL := 45.8;   // Roller center position (mm)
    WheelThreadDiameter : LREAL := 77.47;  // Roller diameter (mm)
    PrintRollerDiameter : LREAL := 446.17; // PrintRoller Diameter, this value is used to calculate linespeed
    MasterVelocity      : LREAL := 1;      // Master axis velocity, this value used to calculate curve time.(rpm, Sheet / min)
    GapOfProduct        : LREAL := 5;      // Distance between products.
    MaxAcceleration     : LREAL := 2000;   // mm/s
    AxisID              : UDINT; 
END_VAR
VAR_OUTPUT
    xAborted : BOOL;
END_VAR
VAR
    StateBehaviour           : CBML.ETrigA;
    arCamPoint_3p               : ARRAY[0..3] OF MC_MotionFunctionPoint;
    arCamPoint_4p               : ARRAY[0..4] OF MC_MotionFunctionPoint;
    uiCalculateFeederCurve   : UINT;
    PrintCircumference       : LREAL;
    MaxMachineLineSpeed      : LREAL;
    MachineLineSpeed         : LREAL;
    MaxSlaveLineSpeed        : LREAL;
    WheelThreadCircumference : LREAL;
    SlaveLineSpeedScale      : LREAL;
    SlaveSyncSpeed           : LREAL;
    SlaveSyncDistance        : LREAL;
    SlaveSyncDistance_deg    : LREAL;
    SlaveSyncTime            : LREAL;
    SlaveSyncTime_deg        : LREAL; // Trans to Master deg
    GapOfProduct_deg         : LREAL;
    SlaveWaitGapTime         : LREAL;
    AccTime                  : LREAL;
    AccTime_deg              : LREAL;
    AccDistance_deg          : LREAL;
    MasterAccDeg             : LREAL;

    // Calculate Curve
    Curve1_MasterPosition : LREAL; // (deg)
    Curve1_SlavePosition  : LREAL; // (mm)
    Curve2_MasterPosition : LREAL; // (deg)
    Curve2_SlavePosition  : LREAL; // (mm)
    Curve2_SlaveVelocity  : LREAL; // (mm/s)
    Curve3_MasterPosition : LREAL; // (deg)
    Curve3_SlavePosition  : LREAL; // (mm)
    Curve4_MasterPosition : LREAL; // (deg)
    Curve4_SlavePosition  : LREAL; // (mm)
	Curve4_active : BOOL;
END_VAR

THIS^.IBehaviourModel := StateBehaviour;
StateBehaviour(
	xExecute:= xExecute, 
	xDone=> xDone, 
	xBusy=> xBusy, 
	xError=> xError, 
	xAbort:= xAbort,
	xAborted=> xAborted);

METHOD CyclicAction
VAR_INPUT
    itfTimingController : CBML.ITimingController;
END_VAR
VAR_OUTPUT
    xComplete : BOOL := TRUE;
    iErrorID : INT := 0;
END_VAR
IF NOT Curve4_active THEN
    arAxisCtrl_gb[AxisID].SyncMode.SyncProfile.CamProfile[ProfileNum].ArraySize   := SIZEOF(arCamPoint_3p);
    arAxisCtrl_gb[AxisID].SyncMode.SyncProfile.CamProfile[ProfileNum].NoOfColumns := 1;
    arAxisCtrl_gb[AxisID].SyncMode.SyncProfile.CamProfile[ProfileNum].NoOfRows    := 4;
    arAxisCtrl_gb[AxisID].SyncMode.SyncProfile.CamProfile[ProfileNum].pArray      := ADR(arCamPoint_3p);
    arAxisCtrl_gb[AxisID].SyncMode.SyncProfile.CamProfile[ProfileNum].TableType   := MC_TABLETYPE_MOTIONFUNCTION;

    arCamPoint_3p[0].FunctionType := MOTIONFUNCTYPE_POLYNOM7_MM;
    arCamPoint_3p[0].MasterPos    := 0;
    arCamPoint_3p[0].SlavePos     := 0;
    arCamPoint_3p[0].PointIndex   := 1;
    arCamPoint_3p[0].PointType    := MOTIONPOINTTYPE_VELOCITY;

    arCamPoint_3p[1].FunctionType := MOTIONFUNCTYPE_POLYNOM1;
    arCamPoint_3p[1].MasterPos    := Curve1_MasterPosition;
    arCamPoint_3p[1].SlavePos     := Curve1_SlavePosition;
    arCamPoint_3p[1].PointIndex   := 2;
    arCamPoint_3p[1].PointType    := MOTIONPOINTTYPE_VELOCITY;

    arCamPoint_3p[2].FunctionType := MOTIONFUNCTYPE_POLYNOM7_MM;
    arCamPoint_3p[2].MasterPos    := Curve2_MasterPosition;
    arCamPoint_3p[2].SlavePos     := Curve2_SlavePosition;
    arCamPoint_3p[2].PointIndex   := 3;
    arCamPoint_3p[2].PointType    := MOTIONPOINTTYPE_VELOCITY;

    arCamPoint_3p[3].FunctionType := MOTIONFUNCTYPE_BESCHLTRAPEZ_VR;
    arCamPoint_3p[3].MasterPos    := Curve3_MasterPosition;
    arCamPoint_3p[3].SlavePos     := Curve3_SlavePosition;
    arCamPoint_3p[3].PointIndex   := 4;
    arCamPoint_3p[3].PointType    := MOTIONPOINTTYPE_REST;
ELSE
    arAxisCtrl_gb[AxisID].SyncMode.SyncProfile.CamProfile[ProfileNum].ArraySize   := SIZEOF(arCamPoint_4p);
    arAxisCtrl_gb[AxisID].SyncMode.SyncProfile.CamProfile[ProfileNum].NoOfColumns := 1;
    arAxisCtrl_gb[AxisID].SyncMode.SyncProfile.CamProfile[ProfileNum].NoOfRows    := 5;
    arAxisCtrl_gb[AxisID].SyncMode.SyncProfile.CamProfile[ProfileNum].pArray      := ADR(arCamPoint_4p);
    arAxisCtrl_gb[AxisID].SyncMode.SyncProfile.CamProfile[ProfileNum].TableType   := MC_TABLETYPE_MOTIONFUNCTION;

    arCamPoint_4p[0].FunctionType := MOTIONFUNCTYPE_POLYNOM7_MM;
    arCamPoint_4p[0].MasterPos    := 0;
    arCamPoint_4p[0].SlavePos     := 0;
    arCamPoint_4p[0].PointIndex   := 1;
    arCamPoint_4p[0].PointType    := MOTIONPOINTTYPE_VELOCITY;

    arCamPoint_4p[1].FunctionType := MOTIONFUNCTYPE_POLYNOM1;
    arCamPoint_4p[1].MasterPos    := Curve1_MasterPosition;
    arCamPoint_4p[1].SlavePos     := Curve1_SlavePosition;
    arCamPoint_4p[1].PointIndex   := 2;
    arCamPoint_4p[1].PointType    := MOTIONPOINTTYPE_VELOCITY;

